(* CODESYS project AlphaController_RECOVERED_2021-01-20T14-59-03.project
   VersionPostfix: -alpha/feature/ezfeed
   Version: 0.9.15.0
   Title: MOAB Prototype
   Author: Ben Hess
   CompiledLibraryCompatibilityVersion: CODESYS V3.5 SP16
   Company: Sharp Packaging

Project tree, tasks and I/O mapping:
  Pro18_1174 : Advantech Control x86 RTE V3, Advantech Co., Ltd., order no. 
      , version 3.5.13.0
    application Application
      libraries: Standard, * (System); VisuDialogs, * (System); Unit Conversion Interfaces, * (Intern); Festo_Motion_FHPP_3, 3.5.7.21 (Festo AG & Co. KG); Serial Communication, 3.5.7.0 (3S - Smart Software Solutions GmbH); Storage, 3.5.7.0 (3S - Smart Software Solutions GmbH); SysPort, 3.5.5.0 (System); Time and Date, 3.5.7.0 (3S - Smart Software Solutions GmbH); SysTime, 3.5.9.0 (System); Network, 3.5.7.0 (3S - Smart Software Solutions GmbH); CIP Object, * (3S - Smart Software Solutions GmbH); CAA Memory Block Manager Extern, * (CAA Technical Workgroup); CmpBitmapPool, * (System); IoDrvModbusBase, 3.5.13.0 (3S - Smart Software Solutions GmbH); SysFile, 3.5.15.0 (System); SysCom, 3.5.15.0 (System); Recipe Management, 3.5.15.0 (System); IoDrvModbus, 3.5.15.0 (3S - Smart Software Solutions GmbH); SysTypes Interfaces, * (System); BASIC, * (OSCAT)
      task MainTask (cyclic, interval 5 ms, priority 0) calls PRG_MainProgram
      task IOUpdate (cyclic, interval 5 ms, priority 1) calls nothing
      function SaveValues [ST]
      Event Handlers/
        function OnlineChangeDone [ST]
        function PrepareShutdown [ST]
        function PrepareOnlineChange [ST]
        function PrepareStop [ST]
        function StartDone [ST]
      Programs/
        program PRG_Bagger [ST]
        function block PRG_ [ST]
        program PRG_MainProgram [ST]
        program Faults [ST]
      function RecallValues [ST]
      Symbols
      global variables HMIData
      Interfaces/
        interface IComponentStatus: Mode, Ready
        interface IFaultHandler: RemoveActiveFault, AddActiveFault
        interface ISupervisor: NotifyMachineFaulted, MakeReady
      RecipeManager
        recipe definition Recipes: HMIData.initiateCycle : BOOL; HMIData.ackAllFaults : BOOL; HMIData.makeReady : BOOL; HMIData.jobLoaded : BOOL; HMIData.stopMachine : BOOL; HMIData.version : STRING; HMIData.inCycle : BOOL; HMIData.batchEnable : BOOL; HMIData.batchSetting : UDINT; HMIData.batchCount : UDINT; HMIData.headCycleCount : UDINT; HMIData.pressureBarOpenDelay : REAL; HMIData.pressureBarCloseDelay : REAL; HMIData.passthroughSetting : REAL; HMIData.passthroughOffset : REAL; HMIData.passthroughPosition : REAL; HMIData.lpaDwell : REAL; HMIData.hpaDwell : REAL; HMIData.sealBarDwell : REAL; HMIData.sealBarTemperatureSetting : UDINT; HMIData.sealBarTemperature : UDINT; HMIData.sealFlattenersPosition : REAL; HMIData.bagSkirtLength : REAL; HMIData.bagLength : REAL; HMIData.bagWidth : REAL; HMIData.bagThickness : REAL; HMIData.bagTensionSetting : REAL; HMIData.bagDropTime : REAL; HMIData.bagForwardSpeed : UDINT; HMIData.bagReverseSpeed : UDINT; HMIData.bagEdgePhotoeyeCovered : BOOL; HMIData.printSpeed : UDINT; HMIData.printLength : REAL; HMIData.printOffset : REAL; HMIData.fillerCountSetting : UDINT; HMIData.fillerCurrentCount : UDINT; HMIData.fillerDropTime : REAL; HMIData.loadPlateDelay : REAL; HMIData.loadPlateDwell : REAL; HMIData.exitConveyorDwell : REAL; HMIData.vacuumDwell : REAL; HMIData.IBDDeflateDwellTime : REAL; HMIData.IBDPackageEjectAssistDelayTime : REAL; HMIData.IBDPackageEjectAssistDwellTime : REAL; HMIData.funnelInUse : BOOL; HMIData.funnelOpenDelay : REAL; HMIData.funnelOpeningTime : REAL; HMIData.funnelClosingTime : REAL; HMIData.externalExitConveyorDwell : REAL; HMIData.barcodeGoodReadCount : UDINT; HMIData.barcodeBadReadCount : UDINT; HMIData.barcodeBadReadFaultSetting : UDINT; HMIData.barcodeStartPosition : REAL; HMIData.barcodeScanDistance : REAL; HMIData.barcodeVerifierInUse : BOOL; HMIData.barcodeLastReadString : STRING(100); HMIData.lastCycleTime : REAL; HMIData.averageCycleTime : REAL; HMIData.resetAverageCycleTime : BOOL; HMIData.bagOpenRetrySetting : INT; HMIData.bagOpenRetryCount : INT; HMIData.bagOpenFeedNewBagSetting : INT; HMIData.bagOpenFeedNewBagCount : INT; HMIData.currentJobID : INT; HMIData.separateBeforeSeal : BOOL; HMIData.activateDemoMode : BOOL; HMIData.printerInUse : BOOL; HMIData.printerInstalled : BOOL; HMIData.lpaDuringBagFeedEnable : BOOL; HMIData.lpaBagEjectAssistEnable : BOOL; HMIData.lpaServiceOn : BOOL; HMIData.lpaServiceOff : BOOL; HMIData.lpaServicePulse : BOOL; HMIData.hpaServiceOn : BOOL; HMIData.hpaServicePulse : BOOL; HMIData.exitConveyorStart : BOOL; HMIData.exitConveyorStop : BOOL; HMIData.exitConveyorJog : BOOL; HMIData.exitConveyorJogTime : TIME; HMIData.exitConveyorStartDwell : BOOL; HMIData.pressureBarService.extendCommand : BOOL; HMIData.pressureBarService.retractCommand : BOOL; HMIData.pressureBarService.exhaustCommand : BOOL; HMIData.pressureBarService.extendedFeedback : BOOL; HMIData.pressureBarService.retractedFeedback : BOOL; HMIData.loadPlateService.extendCommand : BOOL; HMIData.loadPlateService.retractCommand : BOOL; HMIData.loadPlateService.exhaustCommand : BOOL; HMIData.loadPlateService.extendedFeedback : BOOL; HMIData.loadPlateService.retractedFeedback : BOOL; HMIData.forwardLoadPlateService.extendCommand : BOOL; HMIData.forwardLoadPlateService.retractCommand : BOOL; HMIData.forwardLoadPlateService.exhaustCommand : BOOL; HMIData.forwardLoadPlateService.extendedFeedback : BOOL; HMIData.forwardLoadPlateService.retractedFeedback : BOOL; HMIData.rearLoadPlateService.extendCommand : BOOL; HMIData.rearLoadPlateService.retractCommand : BOOL; HMIData.rearLoadPlateService.exhaustCommand : BOOL; HMIData.rearLoadPlateService.extendedFeedback : BOOL; HMIData.rearLoadPlateService.retractedFeedback : BOOL; HMIData.loadShelfService.extendCommand : BOOL; HMIData.loadShelfService.retractCommand : BOOL; HMIData.loadShelfService.exhaustCommand : BOOL; HMIData.loadShelfService.extendedFeedback : BOOL; HMIData.loadShelfService.retractedFeedback : BOOL; HMIData.IBDService.extendCommand : BOOL; HMIData.IBDService.retractCommand : BOOL; HMIData.IBDService.exhaustCommand : BOOL; HMIData.IBDService.extendedFeedback : BOOL; HMIData.IBDService.retractedFeedback : BOOL; HMIData.funnelService.extendCommand : BOOL; HMIData.funnelService.retractCommand : BOOL; HMIData.funnelService.exhaustCommand : BOOL; HMIData.funnelService.extendedFeedback : BOOL; HMIData.funnelService.retractedFeedback : BOOL; HMIData.jogBagForward : BOOL; HMIData.jogBagReverse : BOOL; HMIData.jogPassthroughForward : BOOL; HMIData.jogPassthroughReverse : BOOL; HMIData.sealBarServiceCycle : BOOL; HMIData.sealBarServiceRetract : BOOL; HMIData.sealBarServiceExtend : BOOL; HMIData.bagOpenFingersServiceGrab : BOOL; HMIData.bagOpenFingersServiceRelease : BOOL; HMIData.sealFlattenersServiceRaise : BOOL; HMIData.sealFlattenersServiceLower : BOOL; HMIData.sealFlattenersServiceJogIn : BOOL; HMIData.sealFlattenersServiceJogOut : BOOL; HMIData.sealFlattenersManualPositionSetting : REAL; HMIData.sealFlattenersMoveToManualPos : BOOL; HMIData.passthroughManualPositionSetting : REAL; HMIData.passthroughMoveToManualPos : BOOL; HMIData.factoryTestMode : BOOL; HMIData.vacuumServiceOn : BOOL; HMIData.vacuumServiceOff : BOOL; HMIData.printHeadServiceRaise : BOOL; HMIData.printHeadServiceLower : BOOL; HMIData.externalExitConveyorStart : BOOL; HMIData.externalExitConveyorStop : BOOL; HMIData.externalExitConveyorJog : BOOL; HMIData.externalExitConveyorStartDwell : BOOL; HMIData.triggerBarcodeReaderService : BOOL; HMIData.bofSelection : INT; HMIData.sealFlattenersSelection : INT; HMIData.printerSelection : INT; HMIData.integratedExitConveyorSelection : INT; HMIData.externalExitConveyorSelection : INT; HMIData.packageEjectSelection : INT; HMIData.independentBagDeflatorSelection : INT; HMIData.cycleStartButtonSelection : INT; HMIData.barcodeVerifierSelection : INT; HMIData.baggerModelSelection : INT; HMIData.auxIOConfig.factorySelection : INT; HMIData.auxIOConfig.cfgInputSelection : INT; HMIData.auxIOConfig.cfgOutput1Selection : INT; HMIData.auxIOConfig.cfgOutput2Selection : INT; HMIData.fillerFactorySelection : INT; HMIData.funnelFactorySelection : INT; HMIData.murrIOConfigVersion : INT; HMIData.printerConfigVersion : INT; HMIData.frontFilmFeedMotorConfigVersion : INT; HMIData.rearUnwindMotorConfigVersion : INT; HMIData.sealFlattenerMotorConfigVersion : INT; HMIData.printerRibbonLow.active : BOOL; HMIData.printerNotReady.active : BOOL; HMIData.waitingForPrinter.active : BOOL; HMIData.sealBarNotAtTemperature.active : BOOL; HMIData.recoveryModeActive.active : BOOL; HMIData.jobLoadRequired.active : BOOL; HMIData.baggerNotReady.active : BOOL; HMIData.demoModeIsActive.active : BOOL; HMIData.factoryTestModeActive.active : BOOL; HMIData.machineNotTested.active : BOOL; HMIData.packageEjectGuardRemoved.active : BOOL; HMIData.bagLevelLow.active : BOOL; HMIData.fillerModeCycleStartOnly.active : BOOL; HMIData.baggerInhibited.active : BOOL; HMIData.pressureBarState : STRING; HMIData.baggerCycles.reset : BOOL; HMIData.baggerCycles.count : UDINT; HMIData.bagOpenFingerCycles.reset : BOOL; HMIData.bagOpenFingerCycles.count : UDINT; HMIData.bagsMade.reset : BOOL; HMIData.bagsMade.count : UDINT; HMIData.sealBarCycles.reset : BOOL; HMIData.sealBarCycles.count : UDINT; HMIData.pressureBarCycles.reset : BOOL; HMIData.pressureBarCycles.count : UDINT; HMIData.passthroughChanges.reset : BOOL; HMIData.passthroughChanges.count : UDINT; HMIData.loadPlateCycles.reset : BOOL; HMIData.loadPlateCycles.count : UDINT; HMIData.printerCycles.reset : BOOL; HMIData.printerCycles.count : UDINT; HMIData.motorizedSealFlattenerCycles.reset : BOOL; HMIData.motorizedSealFlattenerCycles.count : UDINT; HMIData.bagOpenRetryTotal.reset : BOOL; HMIData.bagOpenRetryTotal.count : UDINT; HMIData.bagsRejectedTotal.reset : BOOL; HMIData.bagsRejectedTotal.count : UDINT; HMIData.resettableBagsMade.reset : BOOL; HMIData.resettableBagsMade.count : UDINT; HMIData.airFilterClean.target : UDINT; HMIData.airFilterClean.name : STRING; HMIData.airFilterClean.units : STRING; HMIData.airFilterClean.reset : BOOL; HMIData.airFilterClean.count : UDINT; HMIData.driveRollerClean.target : UDINT; HMIData.driveRollerClean.name : STRING; HMIData.driveRollerClean.units : STRING; HMIData.driveRollerClean.reset : BOOL; HMIData.driveRollerClean.count : UDINT; HMIData.printHeadClean.target : UDINT; HMIData.printHeadClean.name : STRING; HMIData.printHeadClean.units : STRING; HMIData.printHeadClean.reset : BOOL; HMIData.printHeadClean.count : UDINT; HMIData.pressureBarGuideShaftGuides.target : UDINT; HMIData.pressureBarGuideShaftGuides.name : STRING; HMIData.pressureBarGuideShaftGuides.units : STRING; HMIData.pressureBarGuideShaftGuides.reset : BOOL; HMIData.pressureBarGuideShaftGuides.count : UDINT; HMIData.pressureBarLeak.iExtended : BOOL; HMIData.pressureBarLeak.iRetracted : BOOL; HMIData.pressureBarLeak.maximumStrokeTime : REAL; HMIData.pressureBarLeak.strokeTime : REAL; HMIData.pressureBarLeak.strokeTimer.IN : BOOL; HMIData.pressureBarLeak.strokeTimer.PT : TIME; HMIData.pressureBarLeak.strokeTimer.Q : BOOL; HMIData.pressureBarLeak.strokeTimer.ET : TIME; HMIData.pressureBarLeak.extendedONS.CLK : BOOL; HMIData.pressureBarLeak.extendedONS.Q : BOOL; HMIData.pressureBarLeak.retractedONS.CLK : BOOL; HMIData.pressureBarLeak.retractedONS.Q : BOOL; HMIData.pressureBarLeak.target : UDINT; HMIData.pressureBarLeak.name : STRING; HMIData.pressureBarLeak.units : STRING; HMIData.pressureBarLeak.reset : BOOL; HMIData.pressureBarLeak.count : UDINT; HMIData.loadPlateLeak.iExtended : BOOL; HMIData.loadPlateLeak.iRetracted : BOOL; HMIData.loadPlateLeak.maximumStrokeTime : REAL; HMIData.loadPlateLeak.strokeTime : REAL; HMIData.loadPlateLeak.strokeTimer.IN : BOOL; HMIData.loadPlateLeak.strokeTimer.PT : TIME; HMIData.loadPlateLeak.strokeTimer.Q : BOOL; HMIData.loadPlateLeak.strokeTimer.ET : TIME; HMIData.loadPlateLeak.extendedONS.CLK : BOOL; HMIData.loadPlateLeak.extendedONS.Q : BOOL; HMIData.loadPlateLeak.retractedONS.CLK : BOOL; HMIData.loadPlateLeak.retractedONS.Q : BOOL; HMIData.loadPlateLeak.target : UDINT; HMIData.loadPlateLeak.name : STRING; HMIData.loadPlateLeak.units : STRING; HMIData.loadPlateLeak.reset : BOOL; HMIData.loadPlateLeak.count : UDINT; HMIData.msfHorizontalMotorTemp.iDriveTemp : DINT; HMIData.msfHorizontalMotorTemp.maxTemp : REAL; HMIData.msfHorizontalMotorTemp.DriveTemp : REAL; HMIData.msfHorizontalMotorTemp.target : UDINT; HMIData.msfHorizontalMotorTemp.name : STRING; HMIData.msfHorizontalMotorTemp.units : STRING; HMIData.msfHorizontalMotorTemp.reset : BOOL; HMIData.msfHorizontalMotorTemp.count : UDINT; HMIData.bagDeliveryMotorTemp.iDriveTemp : DINT; HMIData.bagDeliveryMotorTemp.maxTemp : REAL; HMIData.bagDeliveryMotorTemp.DriveTemp : REAL; HMIData.bagDeliveryMotorTemp.target : UDINT; HMIData.bagDeliveryMotorTemp.name : STRING; HMIData.bagDeliveryMotorTemp.units : STRING; HMIData.bagDeliveryMotorTemp.reset : BOOL; HMIData.bagDeliveryMotorTemp.count : UDINT; HMIData.passthroughMotorTemp.iDriveTemp : DINT; HMIData.passthroughMotorTemp.maxTemp : REAL; HMIData.passthroughMotorTemp.DriveTemp : REAL; HMIData.passthroughMotorTemp.target : UDINT; HMIData.passthroughMotorTemp.name : STRING; HMIData.passthroughMotorTemp.units : STRING; HMIData.passthroughMotorTemp.reset : BOOL; HMIData.passthroughMotorTemp.count : UDINT; HMIData.faultActive : BOOL
      trace Trace (task MainTask): PRG_Bagger.moabHead.pressureBar.electricPressureBarMotor.CRTL_Axis.AckStart, PRG_Bagger.moabHead.pressureBar.electricPressureBarMotor.CRTL_Axis.StartTask, PRG_Bagger.moabHead.pressureBar.electricPressureBarMotor.CRTL_Axis.ActualRecordNo, PRG_Bagger.moabHead.pressureBar.electricPressureBarMotor.CRTL_Axis.RecordNo
    System_Diagnosis : System Diagnosis, Advantech Co., Ltd., version 3.5.13.0
        unmapped channels: System Information
    CIFX_EIP : CIFX-EIP, 3S - Smart Software Solutions GmbH, order no. 1, version 3.5.12.0
        settings: IPAddress = [16#C0,16#A8,16#0A,16#15]; SubnetMask = [16#FF,16#FF,16#FF,16#00]; GatewayAddress = [16#00,16#00,16#00,16#00]; ConfigVersion = 50660608
      FestoManifold : CTEU-EP EtherNetIP bus node, Festo AG & Co. KG, order no. CTEU-EP, version Major Revision=16#2, Minor Revision = 16#2
          settings: INITIALIZED = TRUE; IP address of Target = [16#C0,16#A8,16#0A,16#6E]; Keying.Check Vendor Code = FALSE; Keying.Check Product Code = FALSE; Keying.Check Major Revision = FALSE; Keying.Check Minor Revision = FALSE; RequiredConfigVersion = 50660864; Number of Connections = 1; Connection Settings.Requested packet intervall = 10000 µs; Connection Settings.OT Connection Parameters = 18446; Connection Settings.TO Connection Parameters = 18442; Connection Settings.Connection Flags = 1056; Connection Settings.Connection Path Size = 8; Connection Settings.Config#2 Size = 38; Single Port Inputs 8 bytesParam8.ReadOnly = False; Single Port Inputs 8 bytesParam8.BitSize = 8; Single Port Inputs 8 bytesParam8.DataSize = 1; Single Port Inputs 8 bytesParam9.ReadOnly = False; Single Port Inputs 8 bytesParam9.BitSize = 8; Single Port Inputs 8 bytesParam9.DataSize = 1; Single Port Inputs 8 bytesParam10.ReadOnly = False; Single Port Inputs 8 bytesParam10.BitSize = 8; Single Port Inputs 8 bytesParam10.DataSize = 1; Single Port Inputs 8 bytesParam11.ReadOnly = False; Single Port Inputs 8 bytesParam11.BitSize = 8; Single Port Inputs 8 bytesParam11.DataSize = 1; Single Port Inputs 8 bytesParam12.ReadOnly = False; Single Port Inputs 8 bytesParam12.BitSize = 8; Single Port Inputs 8 bytesParam12.DataSize = 1; Single Port Inputs 8 bytesParam13.ReadOnly = False; Single Port Inputs 8 bytesParam13.BitSize = 8; Single Port Inputs 8 bytesParam13.DataSize = 1; Single Port Inputs 8 bytesParam14.ReadOnly = False; Single Port Inputs 8 bytesParam14.BitSize = 8; Single Port Inputs 8 bytesParam14.DataSize = 1; Single Port Inputs 8 bytesParam15.ReadOnly = False; Single Port Inputs 8 bytesParam15.BitSize = 8; Single Port Inputs 8 bytesParam15.DataSize = 1; Single Port Outputs 8bytesParam8.ReadOnly = False; Single Port Outputs 8bytesParam8.BitSize = 8 ... (119 more)
          output oPBar1Extend : BOOL  // Single Port Outputs 8bytesParam8.Bit0
          output oPbar1Retract : BOOL  // Single Port Outputs 8bytesParam8.Bit1
          output opBar2Extend : BOOL  // Single Port Outputs 8bytesParam8.Bit2
          output opbar2Retract : BOOL  // Single Port Outputs 8bytesParam8.Bit3
          output oSealBarExtend : BOOL  // Single Port Outputs 8bytesParam8.Bit4
          output oSealBarRetract : BOOL  // Single Port Outputs 8bytesParam8.Bit5
          output oLPAOn : BOOL  // Single Port Outputs 8bytesParam8.Bit6
          output oHPAOn : BOOL  // Single Port Outputs 8bytesParam8.Bit7
          output oLoadPlateExtend : BOOL  // Single Port Outputs 8bytesParam9.Bit0
          output oLoadPlateRetract : BOOL  // Single Port Outputs 8bytesParam9.Bit1
          output oBOFUp : BOOL  // Single Port Outputs 8bytesParam9.Bit2
          output oBOFDown : BOOL  // Single Port Outputs 8bytesParam9.Bit3
          output oPrintHeadDown : BOOL  // Single Port Outputs 8bytesParam9.Bit4
          output oPrintHeadUp : BOOL  // Single Port Outputs 8bytesParam9.Bit5
          output oVacOn : BOOL  // Single Port Outputs 8bytesParam9.Bit6
          output oSealFlatUp : BOOL  // Single Port Outputs 8bytesParam10.Bit0
          output oSealFlatDown : BOOL  // Single Port Outputs 8bytesParam10.Bit1
          output oFrontLoadPlateToLoad : BOOL  // Single Port Outputs 8bytesParam10.Bit2
          output oLoadShelfUp : BOOL  // Single Port Outputs 8bytesParam10.Bit4
          output oIBDExtend : BOOL  // Single Port Outputs 8bytesParam10.Bit6
          output oIBDRetract : BOOL  // Single Port Outputs 8bytesParam10.Bit7
          output oFunnelOpen : BOOL  // Single Port Outputs 8bytesParam11.Bit0
          output oFunnelClose : BOOL  // Single Port Outputs 8bytesParam11.Bit1
          unmapped channels: Single Port Inputs 8 bytesParam8, Single Port Inputs 8 bytesParam9, Single Port Inputs 8 bytesParam10, Single Port Inputs 8 bytesParam11, Single Port Inputs 8 bytesParam12, Single Port Inputs 8 bytesParam13, Single Port Inputs 8 bytesParam14, Single Port Inputs 8 bytesParam15, Single Port Outputs 8bytesParam8, Single Port Outputs 8bytesParam9, Single Port Outputs 8bytesParam10, Single Port Outputs 8bytesParam11 ... (4 more)
      MSFMotor : SSM23IP-3EG, Applied Motion Products, Inc, order no. SSM23IP-3EG, version Major Revision=16#3, Minor Revision = 16#3
          settings: INITIALIZED = TRUE; IP address of Target = [16#C0,16#A8,16#0A,16#35]; Keying.Check Device Type = FALSE; Keying.Check Vendor Code = FALSE; Keying.Check Product Code = FALSE; Keying.Check Major Revision = FALSE; Keying.Check Minor Revision = FALSE; RequiredConfigVersion = 50660864; Number of Connections = 1; Connection Settings.Requested packet intervall = 5000 µs; Connection Settings.OT Connection Parameters = 18502; Connection Settings.TO Connection Parameters = 18490; Connection Settings.Connection Flags = 1056; Connection Settings.Connection Path Size = 8; Status Code.ReadOnly = False; Status Code.BitSize = 32; Status Code.DataSize = 4; Alarm Code.ReadOnly = False; Alarm Code.BitSize = 32; Alarm Code.DataSize = 4; Supply Voltage.ReadOnly = False; Supply Voltage.BitSize = 32; Supply Voltage.DataSize = 4; Actual Current.ReadOnly = False; Actual Current.BitSize = 32; Actual Current.DataSize = 4; Drive Temperature.ReadOnly = False; Drive Temperature.BitSize = 32; Drive Temperature.DataSize = 4; Encoder Position.ReadOnly = False; Encoder Position.BitSize = 32; Encoder Position.DataSize = 4; Absolute Position.ReadOnly = False; Absolute Position.BitSize = 32; Absolute Position.DataSize = 4; Position Error.ReadOnly = False; Position Error.BitSize = 32; Position Error.DataSize = 4; Actual Velocity.ReadOnly = False; Actual Velocity.BitSize = 32 ... (245 more)
          input  sealFlattenerHorizontalMotorInputs : DINT  // Status Code
          output sealFlattenerHorizontalMotorOutputs : DINT  // Command Word
          unmapped channels: Alarm Code, Supply Voltage, Actual Current, Drive Temperature, Encoder Position, Absolute Position, Position Error, Actual Velocity, Input Status (extended), Input Status (main), Output Status, Analog Input 1 ... (16 more)
      Panther_PA : WAGO 2759-101 ENIP, WAGO Kontakttechnik GmbH & Co. KG, order no. WagoAppEtherNetIP_Adapter, version Major Revision=16#1, Minor Revision = 16#1 (disabled)
          settings: INITIALIZED = TRUE; IP address of Target = [16#C0,16#A8,16#0A,16#A2]; Keying.Check Minor Revision = FALSE; RequiredConfigVersion = 50660864; Number of Connections = 1; Connection Settings.Requested packet intervall = 5000 µs; Connection Settings.OT Connection Parameters = 18470; Connection Settings.TO Connection Parameters = 18466; Connection Settings.Connection Flags = 1056; Connection Settings.Connection Path Size = 8; Connection Settings.Config#2 Size = 2; Configuration Data = [16#00,16#00]; Heartbeat Multiplier = 1; Port 1 Output Data_Param0.ReadOnly = False; Port 1 Output Data_Param0.BitSize = 8; Port 1 Output Data_Param0.DataSize = 1; Port 1 Output Data_Param1.ReadOnly = False; Port 1 Output Data_Param1.BitSize = 8; Port 1 Output Data_Param1.DataSize = 1; Port 1 Output Data_Param2.ReadOnly = False; Port 1 Output Data_Param2.BitSize = 8; Port 1 Output Data_Param2.DataSize = 1; Port 1 Output Data_Param3.ReadOnly = False; Port 1 Output Data_Param3.BitSize = 8; Port 1 Output Data_Param3.DataSize = 1; Port 1 Output Data_Param4.ReadOnly = False; Port 1 Output Data_Param4.BitSize = 8; Port 1 Output Data_Param4.DataSize = 1; Port 1 Output Data_Param5.ReadOnly = False; Port 1 Output Data_Param5.BitSize = 8; Port 1 Output Data_Param5.DataSize = 1; Port 1 Output Data_Param6.ReadOnly = False; Port 1 Output Data_Param6.BitSize = 8; Port 1 Output Data_Param6.DataSize = 1; Port 1 Output Data_Param7.ReadOnly = False; Port 1 Output Data_Param7.BitSize = 8; Port 1 Output Data_Param7.DataSize = 1; Port 1 Output Data_Param8.ReadOnly = False; Port 1 Output Data_Param8.BitSize = 8; Port 1 Output Data_Param8.DataSize = 1 ... (550 more)
          input  iPAPrintEnginePower : BOOL  // Port 1 Output Data_Param0.Bit0
          input  iPAPrintEngineError : BOOL  // Port 1 Output Data_Param0.Bit1
          input  iPARibbonLow : BOOL  // Port 1 Output Data_Param0.Bit2
          input  iPALabelOut : BOOL  // Port 1 Output Data_Param0.Bit3
          input  iPAOnlineDataReady : BOOL  // Port 1 Output Data_Param0.Bit4
          input  iPARibbonOut : BOOL  // Port 1 Output Data_Param0.Bit5
          input  iPAFaulted : BOOL  // Port 1 Output Data_Param0.Bit7
          input  iPACycleComplete : BOOL  // Port 1 Output Data_Param1.Bit0
          input  iPAApplicatorHome : BOOL  // Port 1 Output Data_Param1.Bit1
          input  iPALowLabels : BOOL  // Port 1 Output Data_Param1.Bit2
          input  iPALOTAR : BOOL  // Port 1 Output Data_Param1.Bit3
          input  iPABypassOn : BOOL  // Port 1 Output Data_Param1.Bit6
          input  iPAHeartbeat : BOOL  // Port 1 Output Data_Param1.Bit7
          output oPATrigger1 : BOOL  // Port 1 Input Data_Param0.Bit0
          output oPAReset : BOOL  // Port 1 Input Data_Param0.Bit2
          output oPABypassEnable : BOOL  // Port 1 Input Data_Param0.Bit3
          unmapped channels: Port 1 Output Data_Param0, Port 1 Output Data_Param1, Port 1 Output Data_Param2, Port 1 Output Data_Param3, Port 1 Output Data_Param4, Port 1 Output Data_Param5, Port 1 Output Data_Param6, Port 1 Output Data_Param7, Port 1 Output Data_Param8, Port 1 Output Data_Param9, Port 1 Output Data_Param10, Port 1 Output Data_Param11 ... (52 more)
      Pbar_ServoEIP : SSM23IP-3EG, Applied Motion Products, Inc, order no. SSM23IP-3EG, version Major Revision=16#3, Minor Revision = 16#3
          settings: INITIALIZED = TRUE; IP address of Target = [16#C0,16#A8,16#0A,16#34]; Keying.Check Vendor Code = FALSE; Keying.Check Product Code = FALSE; Keying.Check Major Revision = FALSE; Keying.Check Minor Revision = FALSE; RequiredConfigVersion = 50660864; Number of Connections = 1; Connection Settings.Requested packet intervall = 5000 µs; Connection Settings.OT Connection Parameters = 18502; Connection Settings.TO Connection Parameters = 18490; Connection Settings.Connection Flags = 1056; Connection Settings.Connection Path Size = 8; Status Code.ReadOnly = False; Status Code.BitSize = 32; Status Code.DataSize = 4; Alarm Code.ReadOnly = False; Alarm Code.BitSize = 32; Alarm Code.DataSize = 4; Supply Voltage.ReadOnly = False; Supply Voltage.BitSize = 32; Supply Voltage.DataSize = 4; Actual Current.ReadOnly = False; Actual Current.BitSize = 32; Actual Current.DataSize = 4; Drive Temperature.ReadOnly = False; Drive Temperature.BitSize = 32; Drive Temperature.DataSize = 4; Encoder Position.ReadOnly = False; Encoder Position.BitSize = 32; Encoder Position.DataSize = 4; Absolute Position.ReadOnly = False; Absolute Position.BitSize = 32; Absolute Position.DataSize = 4; Position Error.ReadOnly = False; Position Error.BitSize = 32; Position Error.DataSize = 4; Actual Velocity.ReadOnly = False; Actual Velocity.BitSize = 32; Actual Velocity.DataSize = 4 ... (244 more)
          input  jawPasstrhoughMotorInputs : DINT  // Status Code
          input  iPassthroughHomeSensorClear : BOOL  // Input Status (main).Bit2
          output jawPasstrhoughMotorOutputs : DINT  // Command Word
          unmapped channels: Alarm Code, Supply Voltage, Actual Current, Drive Temperature, Encoder Position, Absolute Position, Position Error, Actual Velocity, Input Status (extended), Input Status (main), Output Status, Analog Input 1 ... (16 more)
      Cube67_BN_E_V2 : Cube67+ BN-E V2, Murrelektronik GmbH, order no. 56535, version Major Revision=16#2, Minor Revision = 16#5
          settings: INITIALIZED = TRUE; IP address of Target = [16#C0,16#A8,16#0A,16#64]; Keying.Check Vendor Code = FALSE; Keying.Check Product Code = FALSE; Keying.Check Major Revision = FALSE; Keying.Check Minor Revision = FALSE; RequiredConfigVersion = 50660864; Number of Connections = 1; Connection Settings.Requested packet intervall = 5000 µs; Connection Settings.OT Connection Parameters = 18624; Connection Settings.TO Connection Parameters = 18708; Connection Settings.Connection Flags = 1056; Connection Settings.Connection Path Size = 8; Input AssemblyParam0.ReadOnly = False; Input AssemblyParam0.BitSize = 8; Input AssemblyParam0.DataSize = 1; Input AssemblyParam1.ReadOnly = False; Input AssemblyParam1.BitSize = 8; Input AssemblyParam1.DataSize = 1; Input AssemblyParam2.ReadOnly = False; Input AssemblyParam2.BitSize = 8; Input AssemblyParam2.DataSize = 1; Input AssemblyParam3.ReadOnly = False; Input AssemblyParam3.BitSize = 8; Input AssemblyParam3.DataSize = 1; Input AssemblyParam4.ReadOnly = False; Input AssemblyParam4.BitSize = 8; Input AssemblyParam4.DataSize = 1; Input AssemblyParam5.ReadOnly = False; Input AssemblyParam5.BitSize = 8; Input AssemblyParam5.DataSize = 1; Input AssemblyParam6.ReadOnly = False; Input AssemblyParam6.BitSize = 8; Input AssemblyParam6.DataSize = 1; Input AssemblyParam7.ReadOnly = False; Input AssemblyParam7.BitSize = 8; Input AssemblyParam7.DataSize = 1; Input AssemblyParam8.ReadOnly = False; Input AssemblyParam8.BitSize = 8; Input AssemblyParam8.DataSize = 1 ... (4114 more)
          input  iAuxFillerTrigger : BOOL  // Input AssemblyParam29.Bit0
          input  iAuxFillerOK : BOOL  // Input AssemblyParam29.Bit1
          input  iAuxConfigInput : BOOL  // Input AssemblyParam29.Bit2
          input  iFunnelOpened : BOOL  // Input AssemblyParam30.Bit0
          input  iRightPalmButton : BOOL  // Input AssemblyParam30.Bit3
          input  iFunnelClosed : BOOL  // Input AssemblyParam31.Bit0
          input  iLeftPalmButton : BOOL  // Input AssemblyParam31.Bit3
          input  iLoadPlateRetracted : BOOL  // Input AssemblyParam32.Bit0
          input  iLoadShelfRetracted : BOOL  // Input AssemblyParam32.Bit1
          input  iEStopOK : BOOL  // Input AssemblyParam32.Bit2
          input  iFrontLoadPlateRetracted : BOOL  // Input AssemblyParam32.Bit3
          input  iPackageEjectGuardClosed : BOOL  // Input AssemblyParam32.Bit6
          input  iLoadPlateExtended : BOOL  // Input AssemblyParam33.Bit0
          input  iLoadShelfExtended : BOOL  // Input AssemblyParam33.Bit1
          input  iFrontLoadPlateExtended : BOOL  // Input AssemblyParam33.Bit3
          input  iBagsLow : BOOL  // Input AssemblyParam33.Bit5
          input  printerDataReady : BOOL  // Input AssemblyParam35.Bit0
          input  printerEndOfPrint : BOOL  // Input AssemblyParam35.Bit1
          input  printerReady : BOOL  // Input AssemblyParam35.Bit2
          input  iPrinterRibbonEncoder : BOOL  // Input AssemblyParam35.Bit3
          input  iBarcodeReadGood : BOOL  // Input AssemblyParam35.Bit4
          input  iPressureBarRetracted : BOOL  // Input AssemblyParam36.Bit0
          input  iLefttFingerBagPresent : BOOL  // Input AssemblyParam36.Bit2
          input  iPressureBarExtended : BOOL  // Input AssemblyParam37.Bit0
          input  iPressureBarNotObstructed : BOOL  // Input AssemblyParam37.Bit1
          input  iRightFingerBagPresent : BOOL  // Input AssemblyParam37.Bit2
          input  iPowerOffButton : BOOL  // Input AssemblyParam37.Bit3
          input  iHeaterBarTempInputs : BYTE  // Input AssemblyParam38
          input  iMurrSystemState : BYTE  // Input Assembly_Param200
          output oMOMConfig : BYTE  // Output AssemblyParam0
          output oAuxBaggerOK : BOOL  // Output Assembly_Param28.Bit0
          output oAuxConfigOut1 : BOOL  // Output Assembly_Param28.Bit1
          output oAuxReadyForFiller : BOOL  // Output Assembly_Param28.Bit2
          output oAuxConfigOut2 : BOOL  // Output Assembly_Param28.Bit3
          output oSoftStart : BOOL  // Output Assembly_Param32.Bit4
          output oRunExitConveyor : BOOL  // Output Assembly_Param33.Bit2
          output oPrinterStartPrint : BOOL  // Output Assembly_Param34.Bit0
          output oRunPrinterRibbonUnwindMotor : BOOL  // Output Assembly_Param34.Bit1
          output oBarcodeTrigger : BOOL  // Output Assembly_Param34.Bit2
          output oRunExternalExitConveyor : BOOL  // Output Assembly_Param36.Bit1
          output oHMILight : BOOL  // Output Assembly_Param36.Bit3
          output oHeaterPulse : BOOL  // Output Assembly_Param37.Bit4
          unmapped channels: Input AssemblyParam0, Input AssemblyParam1, Input AssemblyParam2, Input AssemblyParam3, Input AssemblyParam4, Input AssemblyParam5, Input AssemblyParam6, Input AssemblyParam7, Input AssemblyParam8, Input AssemblyParam9, Input AssemblyParam10, Input AssemblyParam11 ... (445 more)
      Keyence_BCV : Generic EtherNet/IP device, 3S - Smart Software Solutions GmbH, version 3.5.15.0 (disabled)
          settings: INITIALIZED = TRUE; IP address of Target = [16#C0,16#A8,16#0A,16#A1]; MAC address of Target = [16#00,16#00,16#00,16#00,16#00,16#00]; Keying.Compatibility Bit = FALSE; RequiredConfigVersion = 50660864; Number of Connections = 1; Connection Settings.Requested packet intervall (µs) = 10000; Connection Settings.OT Connection Parameters = 18514; Connection Settings.TO Connection Parameters = 18606; Connection Settings.Connection Flags = 1056; Connection Settings.Connection Path Size = 8; Connection Path = [16#20,16#04,16#24,16#01,16#2C,16#65,16#2C,16#64]; Input_Param0.ReadOnly = False; Input_Param0.BitSize = 8; Input_Param0.DataSize = 1; Input_Param1.ReadOnly = False; Input_Param1.BitSize = 8; Input_Param1.DataSize = 1; Input_Param2.ReadOnly = False; Input_Param2.BitSize = 8; Input_Param2.DataSize = 1; Input_Param3.ReadOnly = False; Input_Param3.BitSize = 8; Input_Param3.DataSize = 1; Input_Param4.ReadOnly = False; Input_Param4.BitSize = 8; Input_Param4.DataSize = 1; Input_Param5.ReadOnly = False; Input_Param5.BitSize = 8; Input_Param5.DataSize = 1; Input_Param6.ReadOnly = False; Input_Param6.BitSize = 8; Input_Param6.DataSize = 1; Input_Param7.ReadOnly = False; Input_Param7.BitSize = 8; Input_Param7.DataSize = 1; Input_Param8.ReadOnly = False; Input_Param8.BitSize = 8; Input_Param8.DataSize = 1; Input_Param9.ReadOnly = False ... (2205 more)
          input  keyenceBCVInputs : BYTE  // Input_Param0
          output keyenceBCVOutputs : BYTE  // Output_Param0
          unmapped channels: Input_Param1, Input_Param2, Input_Param3, Input_Param4, Input_Param5, Input_Param6, Input_Param7, Input_Param8, Input_Param9, Input_Param10, Input_Param11, Input_Param12 ... (234 more)
      IBD_Motor : SSM23IP-3EG, Applied Motion Products, Inc, order no. SSM23IP-3EG, version Major Revision=16#3, Minor Revision = 16#3 (disabled)
          settings: INITIALIZED = TRUE; IP address of Target = [16#C0,16#A8,16#0A,16#39]; MAC address of Target = [16#00,16#00,16#00,16#00,16#00,16#00]; Keying.Check Device Type = FALSE; Keying.Check Vendor Code = FALSE; Keying.Check Product Code = FALSE; Keying.Check Major Revision = FALSE; Keying.Check Minor Revision = FALSE; RequiredConfigVersion = 50660864; Number of Connections = 1; Connection Settings.Requested packet intervall = 10000 µs; Connection Settings.OT Connection Parameters = 18502; Connection Settings.TO Connection Parameters = 18490; Connection Settings.Connection Flags = 1056; Connection Settings.Connection Path Size = 8; Status Code.ReadOnly = False; Status Code.BitSize = 32; Status Code.DataSize = 4; Alarm Code.ReadOnly = False; Alarm Code.BitSize = 32; Alarm Code.DataSize = 4; Supply Voltage.ReadOnly = False; Supply Voltage.BitSize = 32; Supply Voltage.DataSize = 4; Actual Current.ReadOnly = False; Actual Current.BitSize = 32; Actual Current.DataSize = 4; Drive Temperature.ReadOnly = False; Drive Temperature.BitSize = 32; Drive Temperature.DataSize = 4; Encoder Position.ReadOnly = False; Encoder Position.BitSize = 32; Encoder Position.DataSize = 4; Absolute Position.ReadOnly = False; Absolute Position.BitSize = 32; Absolute Position.DataSize = 4; Position Error.ReadOnly = False; Position Error.BitSize = 32; Position Error.DataSize = 4; Actual Velocity.ReadOnly = False ... (246 more)
          input  iIBDMotorEIP : DINT  // Status Code
          output oIBDMotorEIP : DINT  // Command Word
          unmapped channels: Alarm Code, Supply Voltage, Actual Current, Drive Temperature, Encoder Position, Absolute Position, Position Error, Actual Velocity, Input Status (extended), Input Status (main), Output Status, Analog Input 1 ... (16 more)
      Infeed_Conveyor_IO : Advantech - ADAM-6150EI, Advantech Co., Ltd., version Major Revision=16#1, Minor Revision = 16#1 (disabled)
          settings: INITIALIZED = TRUE; IP address of Target = [16#C0,16#A8,16#0A,16#46]; Keying.Check Minor Revision = FALSE; RequiredConfigVersion = 50660864; Number of Connections = 1; Connection Settings.Requested packet intervall = 5000 µs; Connection Settings.OT Connection Parameters = 18440; Connection Settings.TO Connection Parameters = 18436; Connection Settings.Connection Flags = 1056; Connection Settings.Connection Path Size = 8; Heartbeat Multiplier = 1; IO Data (T->O)_Param0.ReadOnly = False; IO Data (T->O)_Param0.BitSize = 8; IO Data (T->O)_Param0.DataSize = 1; IO Data (T->O)_Param1.ReadOnly = False; IO Data (T->O)_Param1.BitSize = 8; IO Data (T->O)_Param1.DataSize = 1; IO Data (O->T)_Param0.ReadOnly = False; IO Data (O->T)_Param0.BitSize = 8; IO Data (O->T)_Param0.DataSize = 1; IO Data (O->T)_Param1.ReadOnly = False; IO Data (O->T)_Param1.BitSize = 8; IO Data (O->T)_Param1.DataSize = 1; IO Data (T->O)_Param0.Name = 'IO Data (T->O)_Param0'; IO Data (T->O)_Param0.HelpString = ''; IO Data (T->O)_Param0.ReadOnly = False; IO Data (T->O)_Param0.BitSize = 8; IO Data (T->O)_Param0.DataSize = 1; IO Data (T->O)_Param0.DataType = 'BYTE'; IO Data (T->O)_Param1.Name = 'IO Data (T->O)_Param1'; IO Data (T->O)_Param1.HelpString = ''; IO Data (T->O)_Param1.ReadOnly = False; IO Data (T->O)_Param1.BitSize = 8; IO Data (T->O)_Param1.DataSize = 1; IO Data (T->O)_Param1.DataType = 'BYTE'; IO Data (O->T)_Param0.Name = 'IO Data (O->T)_Param0'; IO Data (O->T)_Param0.HelpString = ''; IO Data (O->T)_Param0.ReadOnly = False; IO Data (O->T)_Param0.BitSize = 8; IO Data (O->T)_Param0.DataSize = 1 ... (8 more)
          input  iInfeedVFDRunning : BOOL  // IO Data (T->O)_Param0.Bit0
          input  iInfeedVFDNotFaulted : BOOL  // IO Data (T->O)_Param0.Bit1
          input  iInfeedFlightSensor : BOOL  // IO Data (T->O)_Param0.Bit4
          output oRunInfeedVFD : BOOL  // IO Data (O->T)_Param0.Bit0
          output oResetInfeedVFD : BOOL  // IO Data (O->T)_Param0.Bit1
          unmapped channels: IO Data (T->O)_Param0, IO Data (T->O)_Param1, IO Data (O->T)_Param0, IO Data (O->T)_Param1
      Bag_Delivery_Rear_Motor : TSM34IP, Applied Motion Products, Inc, order no. TSM34IP, version Major Revision=16#3, Minor Revision = 16#3
          settings: INITIALIZED = TRUE; IP address of Target = [16#C0,16#A8,16#0A,16#38]; MAC address of Target = [16#00,16#00,16#00,16#00,16#00,16#00]; Keying.Check Device Type = FALSE; Keying.Check Vendor Code = FALSE; Keying.Check Product Code = FALSE; Keying.Check Major Revision = FALSE; Keying.Check Minor Revision = FALSE; RequiredConfigVersion = 50660864; Number of Connections = 1; Connection Settings.Requested packet intervall = 10000 µs; Connection Settings.OT Connection Parameters = 18502; Connection Settings.TO Connection Parameters = 18490; Connection Settings.Connection Flags = 1056; Connection Settings.Connection Path Size = 8; Status Code.ReadOnly = False; Status Code.BitSize = 32; Status Code.DataSize = 4; Alarm Code.ReadOnly = False; Alarm Code.BitSize = 32; Alarm Code.DataSize = 4; Supply Voltage.ReadOnly = False; Supply Voltage.BitSize = 32; Supply Voltage.DataSize = 4; Actual Current.ReadOnly = False; Actual Current.BitSize = 32; Actual Current.DataSize = 4; Drive Temperature.ReadOnly = False; Drive Temperature.BitSize = 32; Drive Temperature.DataSize = 4; Encoder Position.ReadOnly = False; Encoder Position.BitSize = 32; Encoder Position.DataSize = 4; Absolute Position.ReadOnly = False; Absolute Position.BitSize = 32; Absolute Position.DataSize = 4; Position Error.ReadOnly = False; Position Error.BitSize = 32; Position Error.DataSize = 4; Actual Velocity.ReadOnly = False ... (246 more)
          input  bagRearMotorInputs AT %ID200 : DINT  // Status Code
          input  iBagTensionFault : BOOL  // Output Status.Bit3
          output bagRearMotorOutputs AT %QD200 : DINT  // Command Word
          unmapped channels: Alarm Code, Supply Voltage, Actual Current, Drive Temperature, Encoder Position, Absolute Position, Position Error, Actual Velocity, Input Status (extended), Input Status (main), Output Status, Analog Input 1 ... (16 more)
      Bag_Delivery_EIP_Motor : TSM34IP, Applied Motion Products, Inc, order no. TSM34IP, version Major Revision=16#3, Minor Revision = 16#3
          settings: INITIALIZED = TRUE; IP address of Target = [16#C0,16#A8,16#0A,16#37]; Keying.Check Vendor Code = FALSE; Keying.Check Product Code = FALSE; Keying.Check Major Revision = FALSE; Keying.Check Minor Revision = FALSE; RequiredConfigVersion = 50660864; Number of Connections = 1; Connection Settings.Requested packet intervall = 5000 µs; Connection Settings.OT Connection Parameters = 18502; Connection Settings.TO Connection Parameters = 18490; Connection Settings.Connection Flags = 1056; Connection Settings.Connection Path Size = 8; Status Code.ReadOnly = False; Status Code.BitSize = 32; Status Code.DataSize = 4; Alarm Code.ReadOnly = False; Alarm Code.BitSize = 32; Alarm Code.DataSize = 4; Supply Voltage.ReadOnly = False; Supply Voltage.BitSize = 32; Supply Voltage.DataSize = 4; Actual Current.ReadOnly = False; Actual Current.BitSize = 32; Actual Current.DataSize = 4; Drive Temperature.ReadOnly = False; Drive Temperature.BitSize = 32; Drive Temperature.DataSize = 4; Encoder Position.ReadOnly = False; Encoder Position.BitSize = 32; Encoder Position.DataSize = 4; Absolute Position.ReadOnly = False; Absolute Position.BitSize = 32; Absolute Position.DataSize = 4; Position Error.ReadOnly = False; Position Error.BitSize = 32; Position Error.DataSize = 4; Actual Velocity.ReadOnly = False; Actual Velocity.BitSize = 32; Actual Velocity.DataSize = 4 ... (244 more)
          input  bagDeliveryMotorInputs : DINT  // Status Code
          input  iBagNotPresent : BOOL  // Input Status (main).Bit2
          output bagDeliveryMotorOutputs : DINT  // Command Word
          unmapped channels: Alarm Code, Supply Voltage, Actual Current, Drive Temperature, Encoder Position, Absolute Position, Position Error, Actual Velocity, Input Status (extended), Input Status (main), Output Status, Analog Input 1 ... (16 more)
    Ethernet : Ethernet, 3S - Smart Software Solutions GmbH, version 3.5.15.0
        settings: IPAddress = [192,168,10,20]; SubnetMask = [255,255,255,0]; GatewayAddress = [192,168,10,254]; MACAddress = [16#74,16#FE,16#48,16#3F,16#C0,16#65]; NetworkInterfaceName = 'Machine LAN:2'; NetworkInterfaceName = "Machine LAN:2"; SaveCommunicationSettings = FALSE
  ElectricMachine : Advantech Control x86 RTE V3, Advantech Co., Ltd., order no. 
      , version 3.5.16.10
    application Application
      libraries: Standard, * (System); VisuDialogs, * (System); Unit Conversion Interfaces, * (Intern); Festo_Motion_FHPP_3, 3.5.7.21 (Festo AG & Co. KG); Serial Communication, 3.5.7.0 (3S - Smart Software Solutions GmbH); Storage, 3.5.7.0 (3S - Smart Software Solutions GmbH); SysPort, 3.5.5.0 (System); Time and Date, 3.5.7.0 (3S - Smart Software Solutions GmbH); SysTime, 3.5.9.0 (System); Network, 3.5.7.0 (3S - Smart Software Solutions GmbH); CIP Object, * (3S - Smart Software Solutions GmbH); CAA Memory Block Manager Extern, * (CAA Technical Workgroup); CmpBitmapPool, * (System); SysFile, 3.5.15.0 (System); SysCom, 3.5.15.0 (System); Recipe Management, 3.5.15.0 (System); SysTypes Interfaces, * (System); BASIC, * (OSCAT); IoDrvModbusBase, 3.5.16.0 (3S - Smart Software Solutions GmbH); IoDrvModbus, 3.5.16.0 (3S - Smart Software Solutions GmbH)
      task ENIPScannerIOTask (cyclic, interval 5 ms, priority 0) calls EtherNet_IP_Scanner.IOCycle
      task MainTask (cyclic, interval 5 ms, priority 1) calls PRG_MainProgram
      task ENIPScannerServiceTask (cyclic, interval t#20ms, priority 30) calls EtherNet_IP_Scanner.ServiceCycle
      function PrepareShutdown [ST]
      Event Handlers/
        function StartDone [ST]
      Interfaces/
        interface IFaultHandler: AddActiveFault, RemoveActiveFault
        interface IComponentStatus: Mode, Ready
        interface ISupervisor: NotifyMachineFaulted, MakeReady
      RecipeManager
        recipe definition Recipes: HMIData.initiateCycle : BOOL; HMIData.ackAllFaults : BOOL; HMIData.makeReady : BOOL; HMIData.jobLoaded : BOOL; HMIData.stopMachine : BOOL; HMIData.version : STRING; HMIData.inCycle : BOOL; HMIData.batchEnable : BOOL; HMIData.autoEnable : BOOL; HMIData.autoDwell : REAL; HMIData.batchSetting : UDINT; HMIData.batchCount : UDINT; HMIData.headCycleCount : UDINT; HMIData.pressureBarOpenDelay : REAL; HMIData.pressureBarCloseDelay : REAL; HMIData.passthroughSetting : REAL; HMIData.passthroughOffset : REAL; HMIData.passthroughPosition : REAL; HMIData.lpaDwell : REAL; HMIData.hpaDwell : REAL; HMIData.sealBarDwell : REAL; HMIData.sealBarTemperatureSetting : UDINT; HMIData.sealBarTemperature : UDINT; HMIData.sealFlattenersPosition : REAL; HMIData.bagSkirtLength : REAL; HMIData.bagLength : REAL; HMIData.bagWidth : REAL; HMIData.bagThickness : REAL; HMIData.bagTensionSetting : REAL; HMIData.bagDropTime : REAL; HMIData.bagForwardSpeed : UDINT; HMIData.bagReverseSpeed : UDINT; HMIData.bagEdgePhotoeyeCovered : BOOL; HMIData.printSpeed : UDINT; HMIData.printLength : REAL; HMIData.printOffset : REAL; HMIData.fillerCountSetting : UDINT; HMIData.fillerCurrentCount : UDINT; HMIData.fillerDropTime : REAL; HMIData.fillerEnable : BOOL; HMIData.loadPlateDelay : REAL; HMIData.loadPlateDwell : REAL; HMIData.exitConveyorDwell : REAL; HMIData.vacuumDwell : REAL; HMIData.IBDDeflateDwellTime : REAL; HMIData.IBDPackageEjectAssistDelayTime : REAL; HMIData.IBDPackageEjectAssistDwellTime : REAL; HMIData.funnelInUse : BOOL; HMIData.funnelOpenDelay : REAL; HMIData.funnelOpeningTime : REAL; HMIData.funnelClosingTime : REAL; HMIData.externalExitConveyorDwell : REAL; HMIData.barcodeGoodReadCount : UDINT; HMIData.barcodeBadReadCount : UDINT; HMIData.barcodeBadReadFaultSetting : UDINT; HMIData.barcodeStartPosition : REAL; HMIData.barcodeScanDistance : REAL; HMIData.barcodeVerifierInUse : BOOL; HMIData.barcodeLastReadString : STRING(100); HMIData.lastCycleTime : REAL; HMIData.averageCycleTime : REAL; HMIData.resetAverageCycleTime : BOOL; HMIData.bagOpenRetrySetting : INT; HMIData.bagOpenRetryCount : INT; HMIData.bagOpenFeedNewBagSetting : INT; HMIData.bagOpenFeedNewBagCount : INT; HMIData.currentJobID : INT; HMIData.separateBeforeSeal : BOOL; HMIData.activateDemoMode : BOOL; HMIData.printerInUse : BOOL; HMIData.printerInstalled : BOOL; HMIData.lpaDuringBagFeedEnable : BOOL; HMIData.lpaBagEjectAssistEnable : BOOL; HMIData.infeedConveyorRunningMode : BOOL; HMIData.infeedConveyorCountingMode : BOOL; HMIData.infeedIndexDwellTimer : REAL; HMIData.infeedFlightCountTarget : DINT; HMIData.infeedFlightCountActual : DINT; HMIData.infeedPartsCountTarget : DINT; HMIData.infeedPartsCountActual : DINT; HMIData.infeedEmptyPartsSetting : DINT; HMIData.infeedEmptyPartsActual : DINT; HMIData.printAndApplyConveyorDwell : REAL; HMIData.printAndApplyProductToPhotoeyeTime : REAL; HMIData.printAndApplyWaitForLabelTimeout : REAL; HMIData.lpaServiceOn : BOOL; HMIData.lpaServiceOff : BOOL; HMIData.lpaServicePulse : BOOL; HMIData.hpaServiceOn : BOOL; HMIData.hpaServicePulse : BOOL; HMIData.exitConveyorStart : BOOL; HMIData.exitConveyorStop : BOOL; HMIData.exitConveyorJog : BOOL; HMIData.exitConveyorJogTime : TIME; HMIData.exitConveyorStartDwell : BOOL; HMIData.pressureBarService.extendCommand : BOOL; HMIData.pressureBarService.retractCommand : BOOL; HMIData.pressureBarService.exhaustCommand : BOOL; HMIData.pressureBarService.extendedFeedback : BOOL; HMIData.pressureBarService.retractedFeedback : BOOL; HMIData.loadPlateService.extendCommand : BOOL; HMIData.loadPlateService.retractCommand : BOOL; HMIData.loadPlateService.exhaustCommand : BOOL; HMIData.loadPlateService.extendedFeedback : BOOL; HMIData.loadPlateService.retractedFeedback : BOOL; HMIData.forwardLoadPlateService.extendCommand : BOOL; HMIData.forwardLoadPlateService.retractCommand : BOOL; HMIData.forwardLoadPlateService.exhaustCommand : BOOL; HMIData.forwardLoadPlateService.extendedFeedback : BOOL; HMIData.forwardLoadPlateService.retractedFeedback : BOOL; HMIData.rearLoadPlateService.extendCommand : BOOL; HMIData.rearLoadPlateService.retractCommand : BOOL; HMIData.rearLoadPlateService.exhaustCommand : BOOL; HMIData.rearLoadPlateService.extendedFeedback : BOOL; HMIData.rearLoadPlateService.retractedFeedback : BOOL; HMIData.loadShelfService.extendCommand : BOOL; HMIData.loadShelfService.retractCommand : BOOL; HMIData.loadShelfService.exhaustCommand : BOOL; HMIData.loadShelfService.extendedFeedback : BOOL; HMIData.loadShelfService.retractedFeedback : BOOL; HMIData.IBDService.extendCommand : BOOL; HMIData.IBDService.retractCommand : BOOL; HMIData.IBDService.exhaustCommand : BOOL; HMIData.IBDService.extendedFeedback : BOOL; HMIData.IBDService.retractedFeedback : BOOL; HMIData.funnelService.extendCommand : BOOL; HMIData.funnelService.retractCommand : BOOL; HMIData.funnelService.exhaustCommand : BOOL; HMIData.funnelService.extendedFeedback : BOOL; HMIData.funnelService.retractedFeedback : BOOL; HMIData.baggerHeadService.extendCommand : BOOL; HMIData.baggerHeadService.retractCommand : BOOL; HMIData.baggerHeadService.exhaustCommand : BOOL; HMIData.baggerHeadService.extendedFeedback : BOOL; HMIData.baggerHeadService.retractedFeedback : BOOL; HMIData.jogBagForward : BOOL; HMIData.jogBagReverse : BOOL; HMIData.jogPassthroughForward : BOOL; HMIData.jogPassthroughReverse : BOOL; HMIData.sealBarServiceCycle : BOOL; HMIData.sealBarServiceRetract : BOOL; HMIData.sealBarServiceExtend : BOOL; HMIData.bagOpenFingersServiceGrab : BOOL; HMIData.bagOpenFingersServiceRelease : BOOL; HMIData.sealFlattenersServiceRaise : BOOL; HMIData.sealFlattenersServiceLower : BOOL; HMIData.sealFlattenersServiceJogIn : BOOL; HMIData.sealFlattenersServiceJogOut : BOOL; HMIData.sealFlattenersManualPositionSetting : REAL; HMIData.sealFlattenersMoveToManualPos : BOOL; HMIData.passthroughManualPositionSetting : REAL; HMIData.passthroughMoveToManualPos : BOOL; HMIData.factoryTestMode : BOOL; HMIData.vacuumServiceOn : BOOL; HMIData.vacuumServiceOff : BOOL; HMIData.printHeadServiceRaise : BOOL; HMIData.printHeadServiceLower : BOOL; HMIData.externalExitConveyorStart : BOOL; HMIData.externalExitConveyorStop : BOOL; HMIData.externalExitConveyorJog : BOOL; HMIData.externalExitConveyorStartDwell : BOOL; HMIData.triggerBarcodeReaderService : BOOL; HMIData.IBDOffset : REAL; HMIData.bofSelection : INT; HMIData.sealFlattenersSelection : INT; HMIData.printerSelection : INT; HMIData.integratedExitConveyorSelection : INT; HMIData.externalExitConveyorSelection : INT; HMIData.packageEjectSelection : INT; HMIData.independentBagDeflatorSelection : INT; HMIData.cycleStartButtonSelection : INT; HMIData.barcodeVerifierSelection : INT; HMIData.baggerModelSelection : INT; HMIData.auxIOConfig.factorySelection : INT; HMIData.auxIOConfig.cfgInputSelection : INT; HMIData.auxIOConfig.cfgOutput1Selection : INT; HMIData.auxIOConfig.cfgOutput2Selection : INT; HMIData.fillerFactorySelection : INT; HMIData.funnelFactorySelection : INT; HMIData.murrIOConfigVersion : INT; HMIData.printerConfigVersion : INT; HMIData.frontFilmFeedMotorConfigVersion : INT; HMIData.rearUnwindMotorConfigVersion : INT; HMIData.sealFlattenerMotorConfigVersion : INT; HMIData.printerRibbonLow.active : BOOL; HMIData.printerNotReady.active : BOOL; HMIData.waitingForPrinter.active : BOOL; HMIData.sealBarNotAtTemperature.active : BOOL; HMIData.recoveryModeActive.active : BOOL; HMIData.jobLoadRequired.active : BOOL; HMIData.baggerNotReady.active : BOOL; HMIData.demoModeIsActive.active : BOOL; HMIData.factoryTestModeActive.active : BOOL; HMIData.machineNotTested.active : BOOL; HMIData.packageEjectGuardRemoved.active : BOOL; HMIData.bagLevelLow.active : BOOL; HMIData.fillerModeCycleStartOnly.active : BOOL; HMIData.baggerInhibited.active : BOOL; HMIData.infeedConveyorOutOfParts.active : BOOL; HMIData.mayCycleUnexpectedly.active : BOOL; HMIData.printAndApplyRibbonLow.active : BOOL; HMIData.printAndApplyWaitingForApply.active : BOOL; HMIData.printAndApplyWaitingForLabel.active : BOOL; HMIData.printAndApplyBypassed.active : BOOL; HMIData.pressureBarState : STRING; HMIData.baggerCycles.reset : BOOL; HMIData.baggerCycles.count : UDINT; HMIData.bagOpenFingerCycles.reset : BOOL; HMIData.bagOpenFingerCycles.count : UDINT; HMIData.bagsMade.reset : BOOL; HMIData.bagsMade.count : UDINT; HMIData.sealBarCycles.reset : BOOL; HMIData.sealBarCycles.count : UDINT; HMIData.pressureBarCycles.reset : BOOL; HMIData.pressureBarCycles.count : UDINT; HMIData.passthroughChanges.reset : BOOL; HMIData.passthroughChanges.count : UDINT; HMIData.loadPlateCycles.reset : BOOL; HMIData.loadPlateCycles.count : UDINT; HMIData.printerCycles.reset : BOOL; HMIData.printerCycles.count : UDINT; HMIData.motorizedSealFlattenerCycles.reset : BOOL; HMIData.motorizedSealFlattenerCycles.count : UDINT; HMIData.bagOpenRetryTotal.reset : BOOL; HMIData.bagOpenRetryTotal.count : UDINT; HMIData.bagsRejectedTotal.reset : BOOL; HMIData.bagsRejectedTotal.count : UDINT; HMIData.resettableBagsMade.reset : BOOL; HMIData.resettableBagsMade.count : UDINT; HMIData.airFilterClean.target : UDINT; HMIData.airFilterClean.name : STRING; HMIData.airFilterClean.units : STRING; HMIData.airFilterClean.reset : BOOL; HMIData.airFilterClean.count : UDINT; HMIData.driveRollerClean.target : UDINT; HMIData.driveRollerClean.name : STRING; HMIData.driveRollerClean.units : STRING; HMIData.driveRollerClean.reset : BOOL; HMIData.driveRollerClean.count : UDINT; HMIData.printHeadClean.target : UDINT; HMIData.printHeadClean.name : STRING; HMIData.printHeadClean.units : STRING; HMIData.printHeadClean.reset : BOOL; HMIData.printHeadClean.count : UDINT; HMIData.pressureBarGuideShaftGuides.target : UDINT; HMIData.pressureBarGuideShaftGuides.name : STRING; HMIData.pressureBarGuideShaftGuides.units : STRING; HMIData.pressureBarGuideShaftGuides.reset : BOOL; HMIData.pressureBarGuideShaftGuides.count : UDINT; HMIData.pressureBarLeak.iExtended : BOOL; HMIData.pressureBarLeak.iRetracted : BOOL; HMIData.pressureBarLeak.maximumStrokeTime : REAL; HMIData.pressureBarLeak.strokeTime : REAL; HMIData.pressureBarLeak.strokeTimer.IN : BOOL; HMIData.pressureBarLeak.strokeTimer.PT : TIME; HMIData.pressureBarLeak.strokeTimer.Q : BOOL; HMIData.pressureBarLeak.strokeTimer.ET : TIME; HMIData.pressureBarLeak.extendedONS.CLK : BOOL; HMIData.pressureBarLeak.extendedONS.Q : BOOL; HMIData.pressureBarLeak.retractedONS.CLK : BOOL; HMIData.pressureBarLeak.retractedONS.Q : BOOL; HMIData.pressureBarLeak.target : UDINT; HMIData.pressureBarLeak.name : STRING; HMIData.pressureBarLeak.units : STRING; HMIData.pressureBarLeak.reset : BOOL; HMIData.pressureBarLeak.count : UDINT; HMIData.loadPlateLeak.iExtended : BOOL; HMIData.loadPlateLeak.iRetracted : BOOL; HMIData.loadPlateLeak.maximumStrokeTime : REAL; HMIData.loadPlateLeak.strokeTime : REAL; HMIData.loadPlateLeak.strokeTimer.IN : BOOL; HMIData.loadPlateLeak.strokeTimer.PT : TIME; HMIData.loadPlateLeak.strokeTimer.Q : BOOL; HMIData.loadPlateLeak.strokeTimer.ET : TIME; HMIData.loadPlateLeak.extendedONS.CLK : BOOL; HMIData.loadPlateLeak.extendedONS.Q : BOOL; HMIData.loadPlateLeak.retractedONS.CLK : BOOL; HMIData.loadPlateLeak.retractedONS.Q : BOOL; HMIData.loadPlateLeak.target : UDINT; HMIData.loadPlateLeak.name : STRING; HMIData.loadPlateLeak.units : STRING; HMIData.loadPlateLeak.reset : BOOL; HMIData.loadPlateLeak.count : UDINT; HMIData.msfHorizontalMotorTemp.iDriveTemp : DINT; HMIData.msfHorizontalMotorTemp.maxTemp : REAL; HMIData.msfHorizontalMotorTemp.DriveTemp : REAL; HMIData.msfHorizontalMotorTemp.target : UDINT; HMIData.msfHorizontalMotorTemp.name : STRING; HMIData.msfHorizontalMotorTemp.units : STRING; HMIData.msfHorizontalMotorTemp.reset : BOOL; HMIData.msfHorizontalMotorTemp.count : UDINT; HMIData.bagDeliveryMotorTemp.iDriveTemp : DINT; HMIData.bagDeliveryMotorTemp.maxTemp : REAL; HMIData.bagDeliveryMotorTemp.DriveTemp : REAL; HMIData.bagDeliveryMotorTemp.target : UDINT; HMIData.bagDeliveryMotorTemp.name : STRING; HMIData.bagDeliveryMotorTemp.units : STRING; HMIData.bagDeliveryMotorTemp.reset : BOOL; HMIData.bagDeliveryMotorTemp.count : UDINT; HMIData.passthroughMotorTemp.iDriveTemp : DINT; HMIData.passthroughMotorTemp.maxTemp : REAL; HMIData.passthroughMotorTemp.DriveTemp : REAL; HMIData.passthroughMotorTemp.target : UDINT; HMIData.passthroughMotorTemp.name : STRING; HMIData.passthroughMotorTemp.units : STRING; HMIData.passthroughMotorTemp.reset : BOOL; HMIData.passthroughMotorTemp.count : UDINT; HMIData.faultActive : BOOL
      global variables HMIData
      trace Trace (task MainTask): PRG_Bagger.moabHead.pressureBar.electricPressureBarMotor.CRTL_Axis.AckStart, PRG_Bagger.moabHead.pressureBar.electricPressureBarMotor.CRTL_Axis.StartTask, PRG_Bagger.moabHead.pressureBar.electricPressureBarMotor.CRTL_Axis.ActualRecordNo, PRG_Bagger.moabHead.pressureBar.electricPressureBarMotor.CRTL_Axis.RecordNo
      Programs/
        program PRG_Bagger [ST]
        program Faults [ST]
        function block PRG_ [ST]
        program PRG_MainProgram [ST]
      function SaveValues [ST]
      Symbols
      function RecallValues [ST]
      function PrepareStop [ST]
    System_Diagnosis : System Diagnosis, Advantech Co., Ltd., version 3.5.16.10
        unmapped channels: System Information, LED
    Dual_LAN_Card : Ethernet, 3S - Smart Software Solutions GmbH, version 3.5.16.0
        settings: IPAddress = [192,168,10,21]; SubnetMask = [255,255,255,0]; GatewayAddress = [0,0,0,0]; MACAddress = [16#00,16#00,16#00,16#00,16#00,16#00]; NetworkInterfaceName = 'IO Connection'; NetworkInterfaceName = "IO Connection"; SaveCommunicationSettings = FALSE
      EtherNet_IP_Scanner : EtherNet/IP Scanner, 3S - Smart Software Solutions GmbH, order no. 1, version 3.5.16.10
        IBD_Motor : SSM23IP-3EG, Applied Motion Products, Inc, order no. SSM23IP-3EG, version Major Revision=16#3, Minor Revision = 16#3
            settings: INITIALIZED = TRUE; IP address of Target = [16#C0,16#A8,16#0A,16#39]; MAC address of Target = [16#00,16#00,16#00,16#00,16#00,16#00]; Keying.Check Device Type = FALSE; Keying.Check Vendor Code = FALSE; Keying.Check Product Code = FALSE; Keying.Check Major Revision = FALSE; Keying.Check Minor Revision = FALSE; RequiredConfigVersion = 50660864; Number of Connections = 1; Connection Settings.Requested packet intervall = 10000 µs; Connection Settings.OT Connection Parameters = 18502; Connection Settings.TO Connection Parameters = 18490; Connection Settings.Connection Flags = 1056; Connection Settings.Connection Path Size = 8; Status Code.ReadOnly = False; Status Code.BitSize = 32; Status Code.DataSize = 4; Alarm Code.ReadOnly = False; Alarm Code.BitSize = 32; Alarm Code.DataSize = 4; Supply Voltage.ReadOnly = False; Supply Voltage.BitSize = 32; Supply Voltage.DataSize = 4; Actual Current.ReadOnly = False; Actual Current.BitSize = 32; Actual Current.DataSize = 4; Drive Temperature.ReadOnly = False; Drive Temperature.BitSize = 32; Drive Temperature.DataSize = 4; Encoder Position.ReadOnly = False; Encoder Position.BitSize = 32; Encoder Position.DataSize = 4; Absolute Position.ReadOnly = False; Absolute Position.BitSize = 32; Absolute Position.DataSize = 4; Position Error.ReadOnly = False; Position Error.BitSize = 32; Position Error.DataSize = 4; Actual Velocity.ReadOnly = False ... (246 more)
            input  iIBDMotorEIP : DINT  // Status Code
            output oIBDMotorEIP : DINT  // Command Word
            unmapped channels: Alarm Code, Supply Voltage, Actual Current, Drive Temperature, Encoder Position, Absolute Position, Position Error, Actual Velocity, Input Status (extended), Input Status (main), Output Status, Analog Input 1 ... (16 more)
        Cube67_BN_E_V2 : Cube67+ BN-E V2, Murrelektronik GmbH, order no. 56535, version Major Revision=16#2, Minor Revision = 16#5
            settings: INITIALIZED = TRUE; IP address of Target = [16#C0,16#A8,16#0A,16#64]; Keying.Check Vendor Code = FALSE; Keying.Check Product Code = FALSE; Keying.Check Major Revision = FALSE; Keying.Check Minor Revision = FALSE; RequiredConfigVersion = 50660864; Number of Connections = 1; Connection Settings.Requested packet intervall = 5000 µs; Connection Settings.OT Connection Parameters = 18624; Connection Settings.TO Connection Parameters = 18708; Connection Settings.Connection Flags = 1056; Connection Settings.Connection Path Size = 8; Input AssemblyParam0.ReadOnly = False; Input AssemblyParam0.BitSize = 8; Input AssemblyParam0.DataSize = 1; Input AssemblyParam1.ReadOnly = False; Input AssemblyParam1.BitSize = 8; Input AssemblyParam1.DataSize = 1; Input AssemblyParam2.ReadOnly = False; Input AssemblyParam2.BitSize = 8; Input AssemblyParam2.DataSize = 1; Input AssemblyParam3.ReadOnly = False; Input AssemblyParam3.BitSize = 8; Input AssemblyParam3.DataSize = 1; Input AssemblyParam4.ReadOnly = False; Input AssemblyParam4.BitSize = 8; Input AssemblyParam4.DataSize = 1; Input AssemblyParam5.ReadOnly = False; Input AssemblyParam5.BitSize = 8; Input AssemblyParam5.DataSize = 1; Input AssemblyParam6.ReadOnly = False; Input AssemblyParam6.BitSize = 8; Input AssemblyParam6.DataSize = 1; Input AssemblyParam7.ReadOnly = False; Input AssemblyParam7.BitSize = 8; Input AssemblyParam7.DataSize = 1; Input AssemblyParam8.ReadOnly = False; Input AssemblyParam8.BitSize = 8; Input AssemblyParam8.DataSize = 1 ... (4114 more)
            input  iAuxFillerTrigger : BOOL  // Input AssemblyParam29.Bit0
            input  iAuxFillerOK : BOOL  // Input AssemblyParam29.Bit1
            input  iAuxConfigInput : BOOL  // Input AssemblyParam29.Bit2
            input  iFunnelOpened : BOOL  // Input AssemblyParam30.Bit0
            input  iRightPalmButton : BOOL  // Input AssemblyParam30.Bit3
            input  iFunnelClosed : BOOL  // Input AssemblyParam31.Bit0
            input  iLeftPalmButton : BOOL  // Input AssemblyParam31.Bit3
            input  iLoadPlateRetracted : BOOL  // Input AssemblyParam32.Bit0
            input  iLoadShelfRetracted : BOOL  // Input AssemblyParam32.Bit1
            input  iEStopOK : BOOL  // Input AssemblyParam32.Bit2
            input  iFrontLoadPlateRetracted : BOOL  // Input AssemblyParam32.Bit3
            input  iConveyorClear : BOOL  // Input AssemblyParam32.Bit5
            input  iHeadLowered : BOOL  // Input AssemblyParam32.Bit6
            input  iLoadPlateExtended : BOOL  // Input AssemblyParam33.Bit0
            input  iLoadShelfExtended : BOOL  // Input AssemblyParam33.Bit1
            input  iFrontLoadPlateExtended : BOOL  // Input AssemblyParam33.Bit3
            input  iBagsLow : BOOL  // Input AssemblyParam33.Bit5
            input  iHeadRaised : BOOL  // Input AssemblyParam33.Bit6
            input  printerDataReady : BOOL  // Input AssemblyParam35.Bit0
            input  printerEndOfPrint : BOOL  // Input AssemblyParam35.Bit1
            input  printerReady : BOOL  // Input AssemblyParam35.Bit2
            input  iPrinterRibbonEncoder : BOOL  // Input AssemblyParam35.Bit3
            input  iBarcodeReadGood : BOOL  // Input AssemblyParam35.Bit4
            input  iJawClampsExtended : BOOL  // Input AssemblyParam36.Bit0
            input  iLefttFingerBagPresent : BOOL  // Input AssemblyParam36.Bit2
            input  iJawClamped : BOOL  // Input AssemblyParam36.Bit4
            input  iJawClampsRetracted : BOOL  // Input AssemblyParam37.Bit0
            input  iPressureBarNotObstructed : BOOL  // Input AssemblyParam37.Bit1
            input  iRightFingerBagPresent : BOOL  // Input AssemblyParam37.Bit2
            input  iPowerOffButton : BOOL  // Input AssemblyParam37.Bit3
            input  iJawClearToClamp : BOOL  // Input AssemblyParam37.Bit5
            input  iFootSwitch : BOOL  // Input AssemblyParam37.Bit6
            input  iHeaterBarTempInputs : BYTE  // Input AssemblyParam38
            input  iMurrTouchButtonStatus : BYTE  // Input AssemblyParam41
            input  iLightedTouchButton : BOOL  // Input AssemblyParam41.Bit0
            input  iMurrSystemState : BYTE  // Input Assembly_Param200
            output oMOMConfig : BYTE  // Output AssemblyParam0
            output oAuxBaggerOK : BOOL  // Output Assembly_Param28.Bit0
            output oAuxConfigOut1 : BOOL  // Output Assembly_Param28.Bit1
            output oAuxReadyForFiller : BOOL  // Output Assembly_Param28.Bit2
            output oAuxConfigOut2 : BOOL  // Output Assembly_Param28.Bit3
            output oSoftStart : BOOL  // Output Assembly_Param32.Bit4
            output oBaggerHeadMotorDir : BOOL  // Output Assembly_Param32.Bit7
            output oRunExitConveyor : BOOL  // Output Assembly_Param33.Bit2
            output oRunBaggerHeadMotor : BOOL  // Output Assembly_Param33.Bit7
            output oPrinterStartPrint : BOOL  // Output Assembly_Param34.Bit0
            output oRunPrinterRibbonUnwindMotor : BOOL  // Output Assembly_Param34.Bit1
            output oBarcodeTrigger : BOOL  // Output Assembly_Param34.Bit2
            output oRunExternalExitConveyor : BOOL  // Output Assembly_Param36.Bit1
            output oHMILight : BOOL  // Output Assembly_Param36.Bit3
            output oHeaterPulse : BOOL  // Output Assembly_Param37.Bit4
            output oMurrTouchbuttonState : BYTE  // Output Assembly_Param47
            unmapped channels: Input AssemblyParam0, Input AssemblyParam1, Input AssemblyParam2, Input AssemblyParam3, Input AssemblyParam4, Input AssemblyParam5, Input AssemblyParam6, Input AssemblyParam7, Input AssemblyParam8, Input AssemblyParam9, Input AssemblyParam10, Input AssemblyParam11 ... (443 more)
        MSFMotor : SSM23IP-3EG, Applied Motion Products, Inc, order no. SSM23IP-3EG, version Major Revision=16#3, Minor Revision = 16#3
            settings: INITIALIZED = TRUE; IP address of Target = [16#C0,16#A8,16#0A,16#35]; Keying.Check Device Type = FALSE; Keying.Check Vendor Code = FALSE; Keying.Check Product Code = FALSE; Keying.Check Major Revision = FALSE; Keying.Check Minor Revision = FALSE; RequiredConfigVersion = 50660864; Number of Connections = 1; Connection Settings.Requested packet intervall = 5000 µs; Connection Settings.OT Connection Parameters = 18502; Connection Settings.TO Connection Parameters = 18490; Connection Settings.Connection Flags = 1056; Connection Settings.Connection Path Size = 8; Status Code.ReadOnly = False; Status Code.BitSize = 32; Status Code.DataSize = 4; Alarm Code.ReadOnly = False; Alarm Code.BitSize = 32; Alarm Code.DataSize = 4; Supply Voltage.ReadOnly = False; Supply Voltage.BitSize = 32; Supply Voltage.DataSize = 4; Actual Current.ReadOnly = False; Actual Current.BitSize = 32; Actual Current.DataSize = 4; Drive Temperature.ReadOnly = False; Drive Temperature.BitSize = 32; Drive Temperature.DataSize = 4; Encoder Position.ReadOnly = False; Encoder Position.BitSize = 32; Encoder Position.DataSize = 4; Absolute Position.ReadOnly = False; Absolute Position.BitSize = 32; Absolute Position.DataSize = 4; Position Error.ReadOnly = False; Position Error.BitSize = 32; Position Error.DataSize = 4; Actual Velocity.ReadOnly = False; Actual Velocity.BitSize = 32 ... (245 more)
            input  sealFlattenerHorizontalMotorInputs : DINT  // Status Code
            output sealFlattenerHorizontalMotorOutputs : DINT  // Command Word
            unmapped channels: Alarm Code, Supply Voltage, Actual Current, Drive Temperature, Encoder Position, Absolute Position, Position Error, Actual Velocity, Input Status (extended), Input Status (main), Output Status, Analog Input 1 ... (16 more)
        Bag_Delivery_Rear_Motor : TSM34IP, Applied Motion Products, Inc, order no. TSM34IP, version Major Revision=16#3, Minor Revision = 16#3
            settings: INITIALIZED = TRUE; IP address of Target = [16#C0,16#A8,16#0A,16#38]; MAC address of Target = [16#00,16#00,16#00,16#00,16#00,16#00]; Keying.Check Device Type = FALSE; Keying.Check Vendor Code = FALSE; Keying.Check Product Code = FALSE; Keying.Check Major Revision = FALSE; Keying.Check Minor Revision = FALSE; RequiredConfigVersion = 50660864; Number of Connections = 1; Connection Settings.Requested packet intervall = 10000 µs; Connection Settings.OT Connection Parameters = 18502; Connection Settings.TO Connection Parameters = 18490; Connection Settings.Connection Flags = 1056; Connection Settings.Connection Path Size = 8; Status Code.ReadOnly = False; Status Code.BitSize = 32; Status Code.DataSize = 4; Alarm Code.ReadOnly = False; Alarm Code.BitSize = 32; Alarm Code.DataSize = 4; Supply Voltage.ReadOnly = False; Supply Voltage.BitSize = 32; Supply Voltage.DataSize = 4; Actual Current.ReadOnly = False; Actual Current.BitSize = 32; Actual Current.DataSize = 4; Drive Temperature.ReadOnly = False; Drive Temperature.BitSize = 32; Drive Temperature.DataSize = 4; Encoder Position.ReadOnly = False; Encoder Position.BitSize = 32; Encoder Position.DataSize = 4; Absolute Position.ReadOnly = False; Absolute Position.BitSize = 32; Absolute Position.DataSize = 4; Position Error.ReadOnly = False; Position Error.BitSize = 32; Position Error.DataSize = 4; Actual Velocity.ReadOnly = False ... (246 more)
            input  bagRearMotorInputs AT %ID200 : DINT  // Status Code
            input  iBagTensionFault : BOOL  // Output Status.Bit3
            output bagRearMotorOutputs AT %QD200 : DINT  // Command Word
            unmapped channels: Alarm Code, Supply Voltage, Actual Current, Drive Temperature, Encoder Position, Absolute Position, Position Error, Actual Velocity, Input Status (extended), Input Status (main), Output Status, Analog Input 1 ... (16 more)
        Infeed_Conveyor_IO : Advantech - ADAM-6150EI, Advantech Co., Ltd., version Major Revision=16#1, Minor Revision = 16#1 (disabled)
            settings: INITIALIZED = TRUE; IP address of Target = [16#C0,16#A8,16#0A,16#46]; Keying.Check Minor Revision = FALSE; RequiredConfigVersion = 50660864; Number of Connections = 1; Connection Settings.Requested packet intervall = 5000 µs; Connection Settings.OT Connection Parameters = 18440; Connection Settings.TO Connection Parameters = 18436; Connection Settings.Connection Flags = 1056; Connection Settings.Connection Path Size = 8; Heartbeat Multiplier = 1; IO Data (T->O)_Param0.ReadOnly = False; IO Data (T->O)_Param0.BitSize = 8; IO Data (T->O)_Param0.DataSize = 1; IO Data (T->O)_Param1.ReadOnly = False; IO Data (T->O)_Param1.BitSize = 8; IO Data (T->O)_Param1.DataSize = 1; IO Data (O->T)_Param0.ReadOnly = False; IO Data (O->T)_Param0.BitSize = 8; IO Data (O->T)_Param0.DataSize = 1; IO Data (O->T)_Param1.ReadOnly = False; IO Data (O->T)_Param1.BitSize = 8; IO Data (O->T)_Param1.DataSize = 1; IO Data (T->O)_Param0.Name = 'IO Data (T->O)_Param0'; IO Data (T->O)_Param0.HelpString = ''; IO Data (T->O)_Param0.ReadOnly = False; IO Data (T->O)_Param0.BitSize = 8; IO Data (T->O)_Param0.DataSize = 1; IO Data (T->O)_Param0.DataType = 'BYTE'; IO Data (T->O)_Param1.Name = 'IO Data (T->O)_Param1'; IO Data (T->O)_Param1.HelpString = ''; IO Data (T->O)_Param1.ReadOnly = False; IO Data (T->O)_Param1.BitSize = 8; IO Data (T->O)_Param1.DataSize = 1; IO Data (T->O)_Param1.DataType = 'BYTE'; IO Data (O->T)_Param0.Name = 'IO Data (O->T)_Param0'; IO Data (O->T)_Param0.HelpString = ''; IO Data (O->T)_Param0.ReadOnly = False; IO Data (O->T)_Param0.BitSize = 8; IO Data (O->T)_Param0.DataSize = 1 ... (8 more)
            input  iInfeedVFDRunning : BOOL  // IO Data (T->O)_Param0.Bit0
            input  iInfeedVFDNotFaulted : BOOL  // IO Data (T->O)_Param0.Bit1
            input  iInfeedFlightSensor : BOOL  // IO Data (T->O)_Param0.Bit4
            output oRunInfeedVFD : BOOL  // IO Data (O->T)_Param0.Bit0
            output oResetInfeedVFD : BOOL  // IO Data (O->T)_Param0.Bit1
            unmapped channels: IO Data (T->O)_Param0, IO Data (T->O)_Param1, IO Data (O->T)_Param0, IO Data (O->T)_Param1
        FestoManifold : CTEU-EP EtherNetIP bus node, Festo AG & Co. KG, order no. CTEU-EP, version Major Revision=16#2, Minor Revision = 16#2
            settings: INITIALIZED = TRUE; IP address of Target = [16#C0,16#A8,16#0A,16#6E]; Keying.Check Vendor Code = FALSE; Keying.Check Product Code = FALSE; Keying.Check Major Revision = FALSE; Keying.Check Minor Revision = FALSE; RequiredConfigVersion = 50660864; Number of Connections = 1; Connection Settings.Requested packet intervall = 10000 µs; Connection Settings.OT Connection Parameters = 18446; Connection Settings.TO Connection Parameters = 18442; Connection Settings.Connection Flags = 1056; Connection Settings.Connection Path Size = 8; Connection Settings.Config#2 Size = 38; Single Port Inputs 8 bytesParam8.ReadOnly = False; Single Port Inputs 8 bytesParam8.BitSize = 8; Single Port Inputs 8 bytesParam8.DataSize = 1; Single Port Inputs 8 bytesParam9.ReadOnly = False; Single Port Inputs 8 bytesParam9.BitSize = 8; Single Port Inputs 8 bytesParam9.DataSize = 1; Single Port Inputs 8 bytesParam10.ReadOnly = False; Single Port Inputs 8 bytesParam10.BitSize = 8; Single Port Inputs 8 bytesParam10.DataSize = 1; Single Port Inputs 8 bytesParam11.ReadOnly = False; Single Port Inputs 8 bytesParam11.BitSize = 8; Single Port Inputs 8 bytesParam11.DataSize = 1; Single Port Inputs 8 bytesParam12.ReadOnly = False; Single Port Inputs 8 bytesParam12.BitSize = 8; Single Port Inputs 8 bytesParam12.DataSize = 1; Single Port Inputs 8 bytesParam13.ReadOnly = False; Single Port Inputs 8 bytesParam13.BitSize = 8; Single Port Inputs 8 bytesParam13.DataSize = 1; Single Port Inputs 8 bytesParam14.ReadOnly = False; Single Port Inputs 8 bytesParam14.BitSize = 8; Single Port Inputs 8 bytesParam14.DataSize = 1; Single Port Inputs 8 bytesParam15.ReadOnly = False; Single Port Inputs 8 bytesParam15.BitSize = 8; Single Port Inputs 8 bytesParam15.DataSize = 1; Single Port Outputs 8bytesParam8.ReadOnly = False; Single Port Outputs 8bytesParam8.BitSize = 8 ... (119 more)
            output oJawClampExtend : BOOL  // Single Port Outputs 8bytesParam8.Bit0
            output oJawClampRetract : BOOL  // Single Port Outputs 8bytesParam8.Bit1
            output oSealBarExtend : BOOL  // Single Port Outputs 8bytesParam8.Bit2
            output oSealBarRetract : BOOL  // Single Port Outputs 8bytesParam8.Bit3
            output oLPAOn : BOOL  // Single Port Outputs 8bytesParam8.Bit4
            output oHPAOn : BOOL  // Single Port Outputs 8bytesParam8.Bit5
            output oLoadPlateExtend : BOOL  // Single Port Outputs 8bytesParam8.Bit6
            output oLoadPlateRetract : BOOL  // Single Port Outputs 8bytesParam8.Bit7
            output oBOFUp : BOOL  // Single Port Outputs 8bytesParam9.Bit0
            output oBOFDown : BOOL  // Single Port Outputs 8bytesParam9.Bit1
            output oPrintHeadDown : BOOL  // Single Port Outputs 8bytesParam9.Bit2
            output oPrintHeadUp : BOOL  // Single Port Outputs 8bytesParam9.Bit3
            output oVacOn : BOOL  // Single Port Outputs 8bytesParam9.Bit4
            output oSealFlatUp : BOOL  // Single Port Outputs 8bytesParam9.Bit6
            output oSealFlatDown : BOOL  // Single Port Outputs 8bytesParam9.Bit7
            output oFrontLoadPlateToLoad : BOOL  // Single Port Outputs 8bytesParam10.Bit2
            output oFrontLoadPlateToDischarge : BOOL  // Single Port Outputs 8bytesParam10.Bit3
            output oLoadShelfUp : BOOL  // Single Port Outputs 8bytesParam10.Bit4
            output oIBDExtend : BOOL  // Single Port Outputs 8bytesParam10.Bit6
            output oIBDRetract : BOOL  // Single Port Outputs 8bytesParam10.Bit7
            output oFunnelOpen : BOOL  // Single Port Outputs 8bytesParam11.Bit0
            output oFunnelClose : BOOL  // Single Port Outputs 8bytesParam11.Bit1
            unmapped channels: Single Port Inputs 8 bytesParam8, Single Port Inputs 8 bytesParam9, Single Port Inputs 8 bytesParam10, Single Port Inputs 8 bytesParam11, Single Port Inputs 8 bytesParam12, Single Port Inputs 8 bytesParam13, Single Port Inputs 8 bytesParam14, Single Port Inputs 8 bytesParam15, Single Port Outputs 8bytesParam8, Single Port Outputs 8bytesParam9, Single Port Outputs 8bytesParam10, Single Port Outputs 8bytesParam11 ... (4 more)
        Pbar_ServoEIP : SSM23IP-3EG, Applied Motion Products, Inc, order no. SSM23IP-3EG, version Major Revision=16#3, Minor Revision = 16#3
            settings: INITIALIZED = TRUE; IP address of Target = [16#C0,16#A8,16#0A,16#34]; Keying.Check Vendor Code = FALSE; Keying.Check Product Code = FALSE; Keying.Check Major Revision = FALSE; Keying.Check Minor Revision = FALSE; RequiredConfigVersion = 50660864; Number of Connections = 1; Connection Settings.Requested packet intervall = 5000 µs; Connection Settings.OT Connection Parameters = 18502; Connection Settings.TO Connection Parameters = 18490; Connection Settings.Connection Flags = 1056; Connection Settings.Connection Path Size = 8; Status Code.ReadOnly = False; Status Code.BitSize = 32; Status Code.DataSize = 4; Alarm Code.ReadOnly = False; Alarm Code.BitSize = 32; Alarm Code.DataSize = 4; Supply Voltage.ReadOnly = False; Supply Voltage.BitSize = 32; Supply Voltage.DataSize = 4; Actual Current.ReadOnly = False; Actual Current.BitSize = 32; Actual Current.DataSize = 4; Drive Temperature.ReadOnly = False; Drive Temperature.BitSize = 32; Drive Temperature.DataSize = 4; Encoder Position.ReadOnly = False; Encoder Position.BitSize = 32; Encoder Position.DataSize = 4; Absolute Position.ReadOnly = False; Absolute Position.BitSize = 32; Absolute Position.DataSize = 4; Position Error.ReadOnly = False; Position Error.BitSize = 32; Position Error.DataSize = 4; Actual Velocity.ReadOnly = False; Actual Velocity.BitSize = 32; Actual Velocity.DataSize = 4 ... (244 more)
            input  jawPasstrhoughMotorInputs : DINT  // Status Code
            output jawPasstrhoughMotorOutputs : DINT  // Command Word
            unmapped channels: Alarm Code, Supply Voltage, Actual Current, Drive Temperature, Encoder Position, Absolute Position, Position Error, Actual Velocity, Input Status (extended), Input Status (main), Output Status, Analog Input 1 ... (16 more)
        Keyence_BCV : Generic EtherNet/IP device, 3S - Smart Software Solutions GmbH, version 3.5.15.0 (disabled)
            settings: INITIALIZED = TRUE; IP address of Target = [16#C0,16#A8,16#0A,16#A1]; MAC address of Target = [16#00,16#00,16#00,16#00,16#00,16#00]; Keying.Compatibility Bit = FALSE; RequiredConfigVersion = 50660864; Number of Connections = 1; Connection Settings.Requested packet intervall (µs) = 10000; Connection Settings.OT Connection Parameters = 18514; Connection Settings.TO Connection Parameters = 18606; Connection Settings.Connection Flags = 1056; Connection Settings.Connection Path Size = 8; Connection Path = [16#20,16#04,16#24,16#01,16#2C,16#65,16#2C,16#64]; Input_Param0.ReadOnly = False; Input_Param0.BitSize = 8; Input_Param0.DataSize = 1; Input_Param1.ReadOnly = False; Input_Param1.BitSize = 8; Input_Param1.DataSize = 1; Input_Param2.ReadOnly = False; Input_Param2.BitSize = 8; Input_Param2.DataSize = 1; Input_Param3.ReadOnly = False; Input_Param3.BitSize = 8; Input_Param3.DataSize = 1; Input_Param4.ReadOnly = False; Input_Param4.BitSize = 8; Input_Param4.DataSize = 1; Input_Param5.ReadOnly = False; Input_Param5.BitSize = 8; Input_Param5.DataSize = 1; Input_Param6.ReadOnly = False; Input_Param6.BitSize = 8; Input_Param6.DataSize = 1; Input_Param7.ReadOnly = False; Input_Param7.BitSize = 8; Input_Param7.DataSize = 1; Input_Param8.ReadOnly = False; Input_Param8.BitSize = 8; Input_Param8.DataSize = 1; Input_Param9.ReadOnly = False ... (2205 more)
            input  keyenceBCVInputs : BYTE  // Input_Param0
            output keyenceBCVOutputs : BYTE  // Output_Param0
            unmapped channels: Input_Param1, Input_Param2, Input_Param3, Input_Param4, Input_Param5, Input_Param6, Input_Param7, Input_Param8, Input_Param9, Input_Param10, Input_Param11, Input_Param12 ... (234 more)
        Panther_PA : WAGO 2759-101 ENIP, WAGO Kontakttechnik GmbH & Co. KG, order no. WagoAppEtherNetIP_Adapter, version Major Revision=16#1, Minor Revision = 16#1
            settings: INITIALIZED = TRUE; IP address of Target = [16#C0,16#A8,16#0A,16#A2]; Keying.Check Minor Revision = FALSE; RequiredConfigVersion = 50660864; Number of Connections = 1; Connection Settings.Requested packet intervall = 5000 µs; Connection Settings.OT Connection Parameters = 18470; Connection Settings.TO Connection Parameters = 18466; Connection Settings.Connection Flags = 1056; Connection Settings.Connection Path Size = 8; Connection Settings.Config#2 Size = 2; Configuration Data = [16#00,16#00]; Heartbeat Multiplier = 1; Port 1 Output Data_Param0.ReadOnly = False; Port 1 Output Data_Param0.BitSize = 8; Port 1 Output Data_Param0.DataSize = 1; Port 1 Output Data_Param1.ReadOnly = False; Port 1 Output Data_Param1.BitSize = 8; Port 1 Output Data_Param1.DataSize = 1; Port 1 Output Data_Param2.ReadOnly = False; Port 1 Output Data_Param2.BitSize = 8; Port 1 Output Data_Param2.DataSize = 1; Port 1 Output Data_Param3.ReadOnly = False; Port 1 Output Data_Param3.BitSize = 8; Port 1 Output Data_Param3.DataSize = 1; Port 1 Output Data_Param4.ReadOnly = False; Port 1 Output Data_Param4.BitSize = 8; Port 1 Output Data_Param4.DataSize = 1; Port 1 Output Data_Param5.ReadOnly = False; Port 1 Output Data_Param5.BitSize = 8; Port 1 Output Data_Param5.DataSize = 1; Port 1 Output Data_Param6.ReadOnly = False; Port 1 Output Data_Param6.BitSize = 8; Port 1 Output Data_Param6.DataSize = 1; Port 1 Output Data_Param7.ReadOnly = False; Port 1 Output Data_Param7.BitSize = 8; Port 1 Output Data_Param7.DataSize = 1; Port 1 Output Data_Param8.ReadOnly = False; Port 1 Output Data_Param8.BitSize = 8; Port 1 Output Data_Param8.DataSize = 1 ... (550 more)
            input  iPAPrintEnginePower : BOOL  // Port 1 Output Data_Param0.Bit0
            input  iPAPrintEngineError : BOOL  // Port 1 Output Data_Param0.Bit1
            input  iPARibbonLow : BOOL  // Port 1 Output Data_Param0.Bit2
            input  iPALabelOut : BOOL  // Port 1 Output Data_Param0.Bit3
            input  iPAOnlineDataReady : BOOL  // Port 1 Output Data_Param0.Bit4
            input  iPARibbonOut : BOOL  // Port 1 Output Data_Param0.Bit5
            input  iPAFaulted : BOOL  // Port 1 Output Data_Param0.Bit7
            input  iPACycleComplete : BOOL  // Port 1 Output Data_Param1.Bit0
            input  iPAApplicatorHome : BOOL  // Port 1 Output Data_Param1.Bit1
            input  iPALowLabels : BOOL  // Port 1 Output Data_Param1.Bit2
            input  iPALOTAR : BOOL  // Port 1 Output Data_Param1.Bit3
            input  iPABypassOn : BOOL  // Port 1 Output Data_Param1.Bit6
            input  iPAHeartbeat : BOOL  // Port 1 Output Data_Param1.Bit7
            output oPATrigger1 : BOOL  // Port 1 Input Data_Param0.Bit0
            output oPAReset : BOOL  // Port 1 Input Data_Param0.Bit2
            output oPABypassEnable : BOOL  // Port 1 Input Data_Param0.Bit3
            unmapped channels: Port 1 Output Data_Param0, Port 1 Output Data_Param1, Port 1 Output Data_Param2, Port 1 Output Data_Param3, Port 1 Output Data_Param4, Port 1 Output Data_Param5, Port 1 Output Data_Param6, Port 1 Output Data_Param7, Port 1 Output Data_Param8, Port 1 Output Data_Param9, Port 1 Output Data_Param10, Port 1 Output Data_Param11 ... (52 more)
        Bag_Delivery_EIP_Motor : TSM34IP, Applied Motion Products, Inc, order no. TSM34IP, version Major Revision=16#3, Minor Revision = 16#3
            settings: INITIALIZED = TRUE; IP address of Target = [16#C0,16#A8,16#0A,16#37]; Keying.Check Vendor Code = FALSE; Keying.Check Product Code = FALSE; Keying.Check Major Revision = FALSE; Keying.Check Minor Revision = FALSE; RequiredConfigVersion = 50660864; Number of Connections = 1; Connection Settings.Requested packet intervall = 5000 µs; Connection Settings.OT Connection Parameters = 18502; Connection Settings.TO Connection Parameters = 18490; Connection Settings.Connection Flags = 1056; Connection Settings.Connection Path Size = 8; Status Code.ReadOnly = False; Status Code.BitSize = 32; Status Code.DataSize = 4; Alarm Code.ReadOnly = False; Alarm Code.BitSize = 32; Alarm Code.DataSize = 4; Supply Voltage.ReadOnly = False; Supply Voltage.BitSize = 32; Supply Voltage.DataSize = 4; Actual Current.ReadOnly = False; Actual Current.BitSize = 32; Actual Current.DataSize = 4; Drive Temperature.ReadOnly = False; Drive Temperature.BitSize = 32; Drive Temperature.DataSize = 4; Encoder Position.ReadOnly = False; Encoder Position.BitSize = 32; Encoder Position.DataSize = 4; Absolute Position.ReadOnly = False; Absolute Position.BitSize = 32; Absolute Position.DataSize = 4; Position Error.ReadOnly = False; Position Error.BitSize = 32; Position Error.DataSize = 4; Actual Velocity.ReadOnly = False; Actual Velocity.BitSize = 32; Actual Velocity.DataSize = 4 ... (244 more)
            input  bagDeliveryMotorInputs : DINT  // Status Code
            input  iBagNotPresent : BOOL  // Input Status (main).Bit2
            output bagDeliveryMotorOutputs : DINT  // Command Word
            unmapped channels: Alarm Code, Supply Voltage, Actual Current, Drive Temperature, Encoder Position, Absolute Position, Position Error, Actual Velocity, Input Status (extended), Input Status (main), Output Status, Analog Input 1 ... (16 more)
    Ethernet : Ethernet, 3S - Smart Software Solutions GmbH, version 3.5.16.0
        settings: IPAddress = [192,168,10,20]; SubnetMask = [255,255,255,0]; GatewayAddress = [192,168,10,254]; MACAddress = [16#00,16#00,16#00,16#00,16#00,16#00]; NetworkInterfaceName = 'Machine LAN'; NetworkInterfaceName = "Machine LAN"; SaveCommunicationSettings = FALSE
  Project Information/
    function GetVersion [ST]
    function GetCompany [ST]
    function GetTitle [ST]
    function GetTextProperty2 [ST]
    function GetTextProperty [ST]
    function GetBooleanProperty [ST]
    function GetVersionProperty [ST]
    function GetNumberProperty [ST]
  Types/
    data type DEVICE_MODES
    Factoy Selection/
      data type IntegratedConveyorSelection
      data type LabelPrinterSelection
      data type PackageEjectionSelection
      data type ExteralConveyorSelection
      data type BCVSelection
      data type BagDeflatorSelection
      data type SealFlattenerSelection
      data type PalmButtonSelection
      data type BagOpenFingersSelection
      data type AuxiliaryIOSelection
      data type FillerSelection
      data type ModelSelection
      data type FunnelSelection
    data type MODBUS_COMM_TYPE
    data type LoadPlateFaultsType
    data type MotorCommFault
    data type Fault
    data type QX_PROGRAMS
    data type PRINT_SPEEDS
    States/
      data type SOLENOID_TEST_STATES
      data type AMP_EIP_MOVE_INITIAL_STATES
      data type MOVE_MODBUS_COMMAND_STATES
      data type JOG_STATES
      data type PRESSURE_BAR_STATES
      data type VACUUM_PICKER_STATES
      data type OPCODE_MODBUS_COMMAND_STATES
      data type FILLER_STATES
      data type GRABBER_STATES
      data type BCR_STATES
      data type PRINT_AND_APPLY_STATES
      data type EZFEED_STATES_1
      data type PASSTHROUGH_SERVO_STATES
      Head/
        data type TEST_HEAD_STATES
        data type PRINTER_STATES
        data type HEAD_STATES
        data type SEAL_FLATTENER_STATES
        data type SEAL_BAR_STATES
        data type SEAL_SEPARATE_STATES
        data type FINISH_CYCLE_STATES
        data type RELEASE_FEED_STATES
        data type BAG_DELIVERY_STATES
        data type BAG_OPEN_ASSIST_STATES
      MurrIOMOdule/
        data type MOM_STATES
        data type MURR_SYSTEM_STATES
      data type JAW_HOMING_STATES
    HMI Types/
      data type PressureBarHMI
    data type ServiceCommands
    data type ORIENTAL_OPERATION_TYPES
    data type PressureBarFaultsType
    data type IOMasterFaultsType
    data type CylinderFaultsType
    data type ModbusLongType
    AuxIO/
      data type AuxOutputSelection
      data type AuxInputSelection
      data type AuxIOConfiguration
    data type Alarm
    data type FaultType
    data type Warning
    data type StepServoFaultsType
    data type STEP_SERVO_OPCODES
    data type CONFIG_VERSIONS
  FBs/
    DataHandlers/
      function block FB_ModbusDWORD [ST]: HighWord, RawValue, LowWord
      function block ModbusLongHandlerFB [ST]: PackDirect, Pack, Unpack
    Fault/
      function block FB_ONS [ST]
      function block FB_GetTime [ST]
      function block FB_Fault [ST]: Execute, InstanceName, RegisterLogger, Ack, Trigger, FB_Init
      data type LogMessageType
      function block FB_HMIFault [ST]: FB_Init, FB_Reinit, Initialize, InstanceName, Execute
      function block FB_InternalLogger [ST]: InstanceName, AddLogItem
    function block FB_TCPClient [ST]: SendLabel
    Cylinders/
      function block FB_CylinderWithFeedback [ST]: Execute
      interface IThreePositonCylinder: Exhaust
      function block FB_CylinderFaults [ST]
      function block FB_Cylinder [ST]: Retract, Extend, Execute
      function block FB_ThreePositionCylinderWithFeedback [ST]: ResetFault, Exhaust, Execute, Faulted
      interface ICylinder: Extend, Execute, Retract
      function block FB_ThreePositionCylinder [ST]: Exhaust
    function block FB_WriteToFile [ST]
    function block FB_EIPCommsConfigure [ST]: ManualReconfig
    function block FB_PredictiveMaint [ST]
    function block GetTime [ST]
    function block FB_CylinderLeak [ST]
    function block FB_DriveTemp [ST]
    function block TimeLeftFB [ST]
    Components/
      function block PrinterFB_Mode2 [ST]: AutoSendPrintSignal, AutoPrintNow, AutoAckPrintDone, Ready, Mode
      function block BagDeliveryFB_BothMotors [ST]: Ready, ClearCommands, Mode, AutoReverseBag, AutoPrinterDone, AutoWaitForPrinter, AutoStartPrintFeed, AutoFeedBagOut, AutoFeedToEye, AutoPrinterReady
      KeyenceL20FB/
        data type eKeyenceLN20_Error_ID
        function block KeyenceNL20FB [ST]: Ready, Mode
        data type eKeyenceLN20FB_States
      function block MotorizedSealFlattenersFB_BagFeed [ST]: AutoMoveIn, AutoMoveToBagHolding, AutoMoveToHandLoad, Ready, Mode, ClearCommands, AutoMoveToClearance, AutoMoveOut
      function block BarcodeReaderFB [ST]: Trigger, BadRead, GoodRead
      function block BagDeliveryFB [ST]: AutoPrinterDone, AutoFeedToEye, AutoWaitForPrinter, AutoReverseBag, ClearCommands, AutoPrinterReady, Mode, Ready, AutoFeedBagOut, AutoStartPrintFeed
      function block AdjustablePassthroughFB [ST]: MovePassthrough, Ready, Mode, AckRequest, HomeEndStop
      function block FillerFB [ST]: BaggerCycledAndReady, Ready, BaggerCycleInitiated, Mode, Reset
      function block PrinterFB [ST]: AutoSendPrintSignal, AutoPrintNow, Mode, AutoAckPrintDone, Ready
      FB_MurrK50/
        function block FB_MurrK50 [ST]
      DelayDwellFB/
        function block DelayDwellFB [ST]: Reset, ManualOff, ManualOn, Trigger, DwellSetting, DelaySetting
        data type DELAY_DWELL_STATES
      FB_MotorizedPressureBar/
        function block FB_CylinderFeedback [ST]
        data type MotorizedPbarStates
        function block FB_MotorizedPressureBar [ST]: CloseJawNoLatch, OpenJaw, CloseJaw, OpenJawForBagFeed, HomeNow
      function block BagOpenFingersFB [ST]: Release, Grab
      EZFeedFB/
        function block EZFeedFB [ST]: Mode, Ready, Reset
        data type EZFEED_STATES
      function block MotorizedSealFlattenersFB [ST]: ClearCommands, AutoMoveOut, Mode, Ready, AutoMoveToClearance, AutoMoveToBagHolding, AutoMoveIn
      function block PneumaticPressureBarFB_1 [ST]: AutoSealBag, RetractCylinder, AutoOpenJaw, ExhaustCylinder, AutoDoneMovingPassthrough, Mode, ExtendCylinderHighPressure, AutoCloseJaw, Ready, AutoMovingPassthrough, ExtendCylinderLowPressure
      function block FunnelFB [ST]: DelaySetting, CloseNow, OpeningTime, OpenNow, ClosingTime
      FB_MotorizedIBD/
        data type MotorizedIBDStates
        function block FB_MotorizedIBD [ST]: CloseIBD, OpenFull, OpenIBD, RemovePower, HomeNow
      function block PneumaticPressureBarFB [ST]: AutoDoneMovingPassthrough, AutoMovingPassthrough, ExhaustCylinder, Ready, Mode, AutoCloseJaw, ExtendCylinderHighPressure, ExtendCylinderLowPressure, AutoOpenJaw, RetractCylinder, AutoSealBag
      function block ElectricPressureBarFB [ST]: AutoCloseJaw, AutoOpenJaw, Mode, Ready, ClearCommands
      function block PickAndPlaceFB [ST]
      function block BagOpenFingersWithSensorsFB [ST]: CheckIfBagGrabbed
      function block MurrIOFB [ST]: Mode, Ready
      function block BaseComponentFB [ST]: Ready, Reset, Mode
      function block PrintAndApplyFB [ST]: BeginCycle, Reset, Ready, Mode
      function block HeadRaiseLowerFB [ST]
      function block MonostableMultivibratorFB [ST]: DelaySetting, Trigger, ManualOn, ManualOff, DwellSetting
    Motors/
      interface IPositionableMotor: Homing, Moving, InPosition, CurrentPosition, Stop, CommandAcknowledged, HomeNow, MoveToPosition, HomeRequired, MoveDistance
      interface IStoredProgramMotor: ActiveStoredProgramNumber, ExecuteStoredProgram
      Applied Motion/
        function block FB_AppliedMotionBagDeliveryMotor_1 [ST]: SetRearMotorToTorqueMode, SetRearMotorToEncoderFollowing, MoveDistance, StopViaProgram, CommandAcknowledged, SetTorque, Execute, SetRearMotorTorqueValue, MoveDistanceFinal
        Modbus Commands/
          function block FB_SendUserRegistersAppliedMotionTCP [ST]: Execute
          function block FB_SendMoveCommandAppliedMotionRTU [ST]: Execute, CheckIfParSendSuccessful
          function block FB_SendBagMoveAppliedMotionTCP [ST]: Execute
          function block FB_SendMoveCommandAppliedMotionTCP [ST]: Execute
          function block FB_SendOpcodeCommandAppliedMotionTCP [ST]: Execute
          function block FB_SendOpcodeCommandAppliedMotionRTU [ST]: Execute
        function block FB_AppliedMotionStepServoMBBase [ST]: Execute, HomeRequired, CommandAcknowledged, ExecuteStoredProgram, ActiveStoredProgramNumber, MoveDistance, InPosition, HomeNow, Stop, Homing, CurrentPosition, Moving, MoveToPosition
        function block FB_AppliedMotionStepServoEIPPassthrough [ST]: HomeNow, DoneClamping, AllowClamping, Stop, SetPositionLimit, Execute
        DataHandlers/
          function block FB_StepServoAlarms [ST]
          function block FB_StepServoCommands [ST]: Enable, AlarmReset, SendHostCommand, FeedToLength, Clear, StopNormal, IdleState, Disable, StopCrash, SendQAndExecute, FeedToPosition
          function block StepServoStatusFB [ST]
        function block FB_AppliedMotionStepServoEIPPassthrough_1 [ST]: DoneClamping, AllowClamping
        function block FB_AppliedMotionBagDeliveryMotorNoFollowing [ST]: MoveDistance, SetRearMotorToTorqueMode, Execute, SetRearMotorToEncoderFollowing, MoveDistanceFinal, CommandAcknowledged, StopViaProgram
        function block FB_AppliedMotionStepServoTCP [ST]: Stop, MoveToPosition, ExecuteStoredProgram, MoveDistance, HomeNow
        function block FB_AppliedMotionStepServoEIPBase [ST]: Stop, Homing, HomeNow, MoveDistance, CommandAcknowledged, InstanceName, MachineFaulted, MoveToPositionTorque, InPosition, Disable, Enable, ResetEncoderPosition, Execute, HomeRequired, ActiveStoredProgramNumber, Reset, Faulted, MoveToPosition, SetTorque, ExecuteStoredProgram, CurrentPosition, Moving, MoveDistanceTorque
        function block FB_AppliedMotionBagDeliveryMotor [ST]: MoveDistance, SendParameters, MoveDistanceFinal, StopViaProgram
        function block FB_AppliedMotionStepServoEIPBaseQX [ST]: Execute, CommandAcknowledged, HomeNow, HomeRequired, Moving, ActiveStoredProgramNumber, InPosition, MoveDistanceTorque, MachineFaulted, Faulted, MoveToPosition, MoveToPositionTorque, Stop, MoveDistance, CurrentPosition, Homing, Reset, RegisterWithFaultHandler, ExecuteStoredProgram
      Festo/
        function block FB_FestoMotor [ST]: ExecuteStoredProgram, Homing, HomeRequired, CurrentPosition, Execute, CommandAcknowledged, Stop, ActiveStoredProgramNumber, InitDrive, Moving, MoveDistance, InPosition, MoveToPosition, HomeNow
    Temp Sensors/
      function block FB_TemperatureSensor [ST]: TempReadingC, TempReadingF, InstanceName
      function block FB_IFMTempSensor [ST]: Execute
      function block FB_TempController [ST]
      interface ITempSensor: TempReadingF, TempReadingC
    function block FB_HMILight [ST]: BlinkSlow, BlinkFast, TurnOff, TurnOn
    function block FB_FaultHandler [ST]: registerFaultSource
    function block SerialMotorTestFB [ST]
    function block FB_BaggerHeadRaise [ST]
    FunctionalAreas/
      function block FB_MOABHead_Electric [ST]
      function block FB_MOABHead [ST]
    function block FB_CycleCounter [ST]: Increment, Clear, SetCount
  text list GlobalTextList
  Library Information/
    function IsLibReleased [ST]
    function GetLibVersion [ST]
    function GetLibVersionNumber [ST]
  global variables Globals
  text list System
  ObjectHandling/
    interface IExecuteAutomatically: Execute
    function block FB_CollectionHandlerAll [ST]: AddObject
    interface IResettable
    interface IFault: Trigger, Ack
    function block FB_CollectionHandlerLogs [ST]: AddObject
    function block FB_CollectionHandlerLoggable [ST]: RegisterAll, AddObject
    interface IAllObjects: InstanceName
    function block FB_CollectionHandlerInitializable [ST]: InitializeAll, AddObject
    global variables GlobalObjects
    function block FB_CollectionHandlerActiveFaults [ST]: RemoveObject, AckAll, AddObject
    interface ILoggable: RegisterLogger
    interface IInitializable: Initialize
    interface IExhaustable
    interface IFault_1: Ack, Trigger
    function block FB_CollectionHandlerFaults [ST]: AckAll, AddObject
    interface IMachineLogger: AddLogItem
    function block FB_CollectionHandlerExecutable [ST]: ExecuteAll, AddObject
*)

// Types/States/Head/TEST_HEAD_STATES
{attribute 'qualified_only'}
{attribute 'strict'}
TYPE TEST_HEAD_STATES :
(
	Idle := 0,
	Cycling := 10,
	StartHoming := 20,
	Homing := 21,
	HomingComplete := 22,
	MovePassthrough := 30,
	MovingPassthrough := 31,
	MovedPassthrough := 32,
	Fault := 99
);
END_TYPE

// Types/DEVICE_MODES
{attribute 'qualified_only'}
{attribute 'strict'}
TYPE DEVICE_MODES :
(
	Manual := 0,	// Control only from service
	Auto := 1,		// Control only from main Bagger Program
	SemiAuto := 2	// Independent control (like as a test fixture)
);
END_TYPE

// Types/States/SOLENOID_TEST_STATES
{attribute 'qualified_only'}
{attribute 'strict'}
TYPE SOLENOID_TEST_STATES :
(
	Extended := 0,
	Retracted := 1,
	FailedToExtend := 2,
	Idle := 3
);
END_TYPE

// Types/Factoy Selection/IntegratedConveyorSelection
{attribute 'qualified_only'}
{attribute 'strict'}
TYPE IntegratedConveyorSelection :
(
	NotInstalled := 0,
	RearExit := 1
);
END_TYPE

// Types/States/Head/PRINTER_STATES
{attribute 'strict'}
{attribute 'qualified_only'}
TYPE PRINTER_STATES :
(
	Idle := 0,
	WaitingForData := 1,
	DataReady := 2,
	BeginPrintCycle := 3,	
	FeedAtPrintSpeed := 10,
	Printing := 11,
	DonePrinting := 20,
	FeedThrough := 21,
	Ready := 40,
	Fault := 99
);
END_TYPE

// Types/Factoy Selection/LabelPrinterSelection
{attribute 'qualified_only'}
{attribute 'strict'}
TYPE LabelPrinterSelection :
(
	NotInstalled := 0,
	ZebraPrinter203DPI := 1,
	ZebraPrinter300DPI := 2,
	PrintAndApply203DPI := 3,
	PrintAndApply300DPI := 4
);
END_TYPE

// Types/States/AMP_EIP_MOVE_INITIAL_STATES
{attribute 'strict'}
{attribute 'qualified_only'}
TYPE AMP_EIP_MOVE_INITIAL_STATES :
(
	Idle := 0,
	SetOutputOff := 10,
	WaitAfterSettingOutputOff := 11,
	MoveMotor := 12,
	WaitAfterMovingMotor := 13,
	SetOutputOn := 14,
	WaitAfterSettingOutputOn := 15,
	Fault := 99
);
END_TYPE

// Types/MODBUS_COMM_TYPE
{attribute 'strict'}
{attribute 'qualified_only'}
TYPE MODBUS_COMM_TYPE :
(
	ModbusTCP := 0,
	ModbusRTU := 1
);
END_TYPE

// Types/AuxIO/AuxOutputSelection
{attribute 'qualified_only'}
{attribute 'strict'}
TYPE AuxOutputSelection :
(
	NotConfigured := 0,
	PrinterDataReady := 1,
	WaitingForPrinter := 2,
	CycleComplete := 3,
	BagMade := 4,
	BagMadePlusLabelRequired := 5,
	BagsLow := 6
);
END_TYPE

// Types/LoadPlateFaultsType
TYPE LoadPlateFaultsType :
STRUCT
	failedToDischarge : FB_Fault(name := 'Failed to Discharge');        // Load Plate failed to reach Discharge Position
    failedToLoad : FB_Fault(name := 'Failed to Load');  // Load Plate failed to reach Loading Position
	sensorFault : FB_Fault(name := 'Failed to Sensor Fault');		// Both sensors active at the same time
END_STRUCT
END_TYPE

// Types/States/MOVE_MODBUS_COMMAND_STATES
{attribute 'strict'}
{attribute 'qualified_only'}
TYPE MOVE_MODBUS_COMMAND_STATES :
(
	Idle := 0,
	SendParameters := 10,
	WaitAfterParametersSent := 11,
	SendOpcode := 20,
	WaitAfterOpcodeSent := 21,
	SendCommand := 31,
	WaitAfterCommandSent := 32,
	SendClearCommand := 40,
	WaitAfterSendClearCommand := 41,
	Fault := 99
);
END_TYPE

// Types/MotorCommFault
TYPE MotorCommFault :
STRUCT
	timeOfFault : DATE_AND_TIME;
	message : STRING;
END_STRUCT
END_TYPE

// Types/Factoy Selection/PackageEjectionSelection
{attribute 'qualified_only'}
{attribute 'strict'}
TYPE PackageEjectionSelection :
(
	NotInstalled := 0,
	RearRetractingLoadPlate := 1,
	LabelSideUp := 2
);
END_TYPE

